//   PLC/PLC Instance <-> EtherCAT Master BKCUCX/TcTerminals210_EK1100_1/TcTerminals210_1BK1250/A_0187(KL 2012, 2 Ch. Output (24V, 0.5 A))
//     PlcTask Outputs/GVL_iXlinker.EtherCAT_Master_BKCUCX.TcTerminals210_EK1100_1.TcTerminals210_1BK1250.A_0187_KL_2012_2_Ch_Output_24V_0_5_A.Channel_1.Output <-> Channel 1/Output
//     PlcTask Outputs/GVL_iXlinker.EtherCAT_Master_BKCUCX.TcTerminals210_EK1100_1.TcTerminals210_1BK1250.A_0187_KL_2012_2_Ch_Output_24V_0_5_A.Channel_2.Output <-> Channel 2/Output
//   PLC/PLC Instance <-> EtherCAT Master BKCUCX/TcTerminals210_EK1100_1/TcTerminals210_1BK1250/A_0188(KL 2022, 2 Ch. Output (24V, 2.0 A))
//     PlcTask Outputs/GVL_iXlinker.EtherCAT_Master_BKCUCX.TcTerminals210_EK1100_1.TcTerminals210_1BK1250.A_0188_KL_2022_2_Ch_Output_24V_2_0_A.Channel_1.Output <-> Channel 1/Output
//     PlcTask Outputs/GVL_iXlinker.EtherCAT_Master_BKCUCX.TcTerminals210_EK1100_1.TcTerminals210_1BK1250.A_0188_KL_2022_2_Ch_Output_24V_2_0_A.Channel_2.Output <-> Channel 2/Output
//   PLC/PLC Instance <-> EtherCAT Master BKCUCX/TcTerminals210_EK1100_1/TcTerminals210_1BK1250/A_0189(KL 2032, 2 Ch. Output with Protection (24V, 0.5 A))
//     PlcTask Outputs/GVL_iXlinker.EtherCAT_Master_BKCUCX.TcTerminals210_EK1100_1.TcTerminals210_1BK1250.A_0189_KL_2032_2_Ch_Output_with_Protection_24V_0_5_A.Channel_1.Output <-> Channel 1/Output
//     PlcTask Outputs/GVL_iXlinker.EtherCAT_Master_BKCUCX.TcTerminals210_EK1100_1.TcTerminals210_1BK1250.A_0189_KL_2032_2_Ch_Output_with_Protection_24V_0_5_A.Channel_2.Output <-> Channel 2/Output
//   PLC/PLC Instance <-> EtherCAT Master BKCUCX/TcTerminals210_EK1100_1/TcTerminals210_1BK1250/A_0190(KL 2114, 4 Ch. Output (24V, 0.5 A))
//     PlcTask Outputs/GVL_iXlinker.EtherCAT_Master_BKCUCX.TcTerminals210_EK1100_1.TcTerminals210_1BK1250.A_0190_KL_2114_4_Ch_Output_24V_0_5_A.Channel_1.Output <-> Channel 1/Output
//     PlcTask Outputs/GVL_iXlinker.EtherCAT_Master_BKCUCX.TcTerminals210_EK1100_1.TcTerminals210_1BK1250.A_0190_KL_2114_4_Ch_Output_24V_0_5_A.Channel_2.Output <-> Channel 2/Output
//     PlcTask Outputs/GVL_iXlinker.EtherCAT_Master_BKCUCX.TcTerminals210_EK1100_1.TcTerminals210_1BK1250.A_0190_KL_2114_4_Ch_Output_24V_0_5_A.Channel_3.Output <-> Channel 3/Output
//     PlcTask Outputs/GVL_iXlinker.EtherCAT_Master_BKCUCX.TcTerminals210_EK1100_1.TcTerminals210_1BK1250.A_0190_KL_2114_4_Ch_Output_24V_0_5_A.Channel_4.Output <-> Channel 4/Output
//   PLC/PLC Instance <-> EtherCAT Master BKCUCX/TcTerminals210_EK1100_1/TcTerminals210_1BK1250/A_0191(KL 2124, 4 Ch. Output (5V, 20 mA))
//     PlcTask Outputs/GVL_iXlinker.EtherCAT_Master_BKCUCX.TcTerminals210_EK1100_1.TcTerminals210_1BK1250.A_0191_KL_2124_4_Ch_Output_5V_20_mA.Channel_1.Output <-> Channel 1/Output
//     PlcTask Outputs/GVL_iXlinker.EtherCAT_Master_BKCUCX.TcTerminals210_EK1100_1.TcTerminals210_1BK1250.A_0191_KL_2124_4_Ch_Output_5V_20_mA.Channel_2.Output <-> Channel 2/Output
//     PlcTask Outputs/GVL_iXlinker.EtherCAT_Master_BKCUCX.TcTerminals210_EK1100_1.TcTerminals210_1BK1250.A_0191_KL_2124_4_Ch_Output_5V_20_mA.Channel_3.Output <-> Channel 3/Output
//     PlcTask Outputs/GVL_iXlinker.EtherCAT_Master_BKCUCX.TcTerminals210_EK1100_1.TcTerminals210_1BK1250.A_0191_KL_2124_4_Ch_Output_5V_20_mA.Channel_4.Output <-> Channel 4/Output
//   PLC/PLC Instance <-> EtherCAT Master BKCUCX/TcTerminals210_EK1100_1/TcTerminals210_1BK1250/A_0192(KL 2134, 4 Ch. Output with Protection (24V, 0.5 A))
//     PlcTask Outputs/GVL_iXlinker.EtherCAT_Master_BKCUCX.TcTerminals210_EK1100_1.TcTerminals210_1BK1250.A_0192_KL_2134_4_Ch_Output_with_Protection_24V_0_5_A.Channel_1.Output <-> Channel 1/Output
//     PlcTask Outputs/GVL_iXlinker.EtherCAT_Master_BKCUCX.TcTerminals210_EK1100_1.TcTerminals210_1BK1250.A_0192_KL_2134_4_Ch_Output_with_Protection_24V_0_5_A.Channel_2.Output <-> Channel 2/Output
//     PlcTask Outputs/GVL_iXlinker.EtherCAT_Master_BKCUCX.TcTerminals210_EK1100_1.TcTerminals210_1BK1250.A_0192_KL_2134_4_Ch_Output_with_Protection_24V_0_5_A.Channel_3.Output <-> Channel 3/Output
//     PlcTask Outputs/GVL_iXlinker.EtherCAT_Master_BKCUCX.TcTerminals210_EK1100_1.TcTerminals210_1BK1250.A_0192_KL_2134_4_Ch_Output_with_Protection_24V_0_5_A.Channel_4.Output <-> Channel 4/Output
//   PLC/PLC Instance <-> EtherCAT Master BKCUCX/TcTerminals210_EK1100_1/TcTerminals210_1BK1250/A_0193(KL 2184, 4 Ch. Output neg. (24V, 0.5 A))
//     PlcTask Outputs/GVL_iXlinker.EtherCAT_Master_BKCUCX.TcTerminals210_EK1100_1.TcTerminals210_1BK1250.A_0193_KL_2184_4_Ch_Output_neg_24V_0_5_A.Channel_1.Output <-> Channel 1/Output
//     PlcTask Outputs/GVL_iXlinker.EtherCAT_Master_BKCUCX.TcTerminals210_EK1100_1.TcTerminals210_1BK1250.A_0193_KL_2184_4_Ch_Output_neg_24V_0_5_A.Channel_2.Output <-> Channel 2/Output
//     PlcTask Outputs/GVL_iXlinker.EtherCAT_Master_BKCUCX.TcTerminals210_EK1100_1.TcTerminals210_1BK1250.A_0193_KL_2184_4_Ch_Output_neg_24V_0_5_A.Channel_3.Output <-> Channel 3/Output
//     PlcTask Outputs/GVL_iXlinker.EtherCAT_Master_BKCUCX.TcTerminals210_EK1100_1.TcTerminals210_1BK1250.A_0193_KL_2184_4_Ch_Output_neg_24V_0_5_A.Channel_4.Output <-> Channel 4/Output
//   PLC/PLC Instance <-> EtherCAT Master BKCUCX/TcTerminals210_EK1100_1/TcTerminals210_1BK1250/A_0194(KL 2212, 2 Ch. Output (24V, 0.5 A with Diag))
//     PlcTask Inputs/GVL_iXlinker.EtherCAT_Master_BKCUCX.TcTerminals210_EK1100_1.TcTerminals210_1BK1250.A_0194_KL_2212_2_Ch_Output_24V_0_5_A_with_Diag.Channel_1.WireBreak <-> Channel 1/WireBreak
//     PlcTask Inputs/GVL_iXlinker.EtherCAT_Master_BKCUCX.TcTerminals210_EK1100_1.TcTerminals210_1BK1250.A_0194_KL_2212_2_Ch_Output_24V_0_5_A_with_Diag.Channel_2.WireBreak <-> Channel 2/WireBreak
//     PlcTask Inputs/GVL_iXlinker.EtherCAT_Master_BKCUCX.TcTerminals210_EK1100_1.TcTerminals210_1BK1250.A_0194_KL_2212_2_Ch_Output_24V_0_5_A_with_Diag.Channel_1.Curcuit <-> Channel 1/Curcuit
//     PlcTask Inputs/GVL_iXlinker.EtherCAT_Master_BKCUCX.TcTerminals210_EK1100_1.TcTerminals210_1BK1250.A_0194_KL_2212_2_Ch_Output_24V_0_5_A_with_Diag.Channel_2.Curcuit <-> Channel 2/Curcuit
//     PlcTask Outputs/GVL_iXlinker.EtherCAT_Master_BKCUCX.TcTerminals210_EK1100_1.TcTerminals210_1BK1250.A_0194_KL_2212_2_Ch_Output_24V_0_5_A_with_Diag.Channel_1.Output <-> Channel 1/Output
//     PlcTask Outputs/GVL_iXlinker.EtherCAT_Master_BKCUCX.TcTerminals210_EK1100_1.TcTerminals210_1BK1250.A_0194_KL_2212_2_Ch_Output_24V_0_5_A_with_Diag.Channel_2.Output <-> Channel 2/Output
//   PLC/PLC Instance <-> EtherCAT Master BKCUCX/TcTerminals210_EK1100_1/TcTerminals210_1BK1250/A_0195(KL 1202, 2 Ch. Input (24V, with Power))
//     PlcTask Inputs/GVL_iXlinker.EtherCAT_Master_BKCUCX.TcTerminals210_EK1100_1.TcTerminals210_1BK1250.A_0195_KL_1202_2_Ch_Input_24V_with_Power.Channel_1.Input <-> Channel 1/Input
//     PlcTask Inputs/GVL_iXlinker.EtherCAT_Master_BKCUCX.TcTerminals210_EK1100_1.TcTerminals210_1BK1250.A_0195_KL_1202_2_Ch_Input_24V_with_Power.Channel_2.Input <-> Channel 2/Input
//     PlcTask Inputs/GVL_iXlinker.EtherCAT_Master_BKCUCX.TcTerminals210_EK1100_1.TcTerminals210_1BK1250.A_0195_KL_1202_2_Ch_Input_24V_with_Power.Channel_1.Error <-> Channel 1/Error
//     PlcTask Inputs/GVL_iXlinker.EtherCAT_Master_BKCUCX.TcTerminals210_EK1100_1.TcTerminals210_1BK1250.A_0195_KL_1202_2_Ch_Input_24V_with_Power.Channel_2.Error <-> Channel 2/Error
//     PlcTask Outputs/GVL_iXlinker.EtherCAT_Master_BKCUCX.TcTerminals210_EK1100_1.TcTerminals210_1BK1250.A_0195_KL_1202_2_Ch_Input_24V_with_Power.Channel_1.Power <-> Channel 1/Power
//     PlcTask Outputs/GVL_iXlinker.EtherCAT_Master_BKCUCX.TcTerminals210_EK1100_1.TcTerminals210_1BK1250.A_0195_KL_1202_2_Ch_Input_24V_with_Power.Channel_2.Power <-> Channel 2/Power
//   PLC/PLC Instance <-> EtherCAT Master BKCUCX/TcTerminals210_EK1100_1/TcTerminals210_1BK1250/A_0196(KL 2404, 4 Ch. Output with Protection (24V, 0.5 A, 2 wire))
//     PlcTask Outputs/GVL_iXlinker.EtherCAT_Master_BKCUCX.TcTerminals210_EK1100_1.TcTerminals210_1BK1250.A_0196_KL_2404_4_Ch_Output_with_Protection_24V_0_5_A_2_wire.Channel_1.Output <-> Channel 1/Output
//     PlcTask Outputs/GVL_iXlinker.EtherCAT_Master_BKCUCX.TcTerminals210_EK1100_1.TcTerminals210_1BK1250.A_0196_KL_2404_4_Ch_Output_with_Protection_24V_0_5_A_2_wire.Channel_2.Output <-> Channel 2/Output
//     PlcTask Outputs/GVL_iXlinker.EtherCAT_Master_BKCUCX.TcTerminals210_EK1100_1.TcTerminals210_1BK1250.A_0196_KL_2404_4_Ch_Output_with_Protection_24V_0_5_A_2_wire.Channel_3.Output <-> Channel 3/Output
//     PlcTask Outputs/GVL_iXlinker.EtherCAT_Master_BKCUCX.TcTerminals210_EK1100_1.TcTerminals210_1BK1250.A_0196_KL_2404_4_Ch_Output_with_Protection_24V_0_5_A_2_wire.Channel_4.Output <-> Channel 4/Output
//   PLC/PLC Instance <-> EtherCAT Master BKCUCX/TcTerminals210_EK1100_1/TcTerminals210_1BK1250/A_0197(KL 2408, 8 Ch. Output (24V, 0.5 A, 3 A max))
//     PlcTask Outputs/GVL_iXlinker.EtherCAT_Master_BKCUCX.TcTerminals210_EK1100_1.TcTerminals210_1BK1250.A_0197_KL_2408_8_Ch_Output_24V_0_5_A_3_A_max.Channel_1.Output <-> Channel 1/Output
//     PlcTask Outputs/GVL_iXlinker.EtherCAT_Master_BKCUCX.TcTerminals210_EK1100_1.TcTerminals210_1BK1250.A_0197_KL_2408_8_Ch_Output_24V_0_5_A_3_A_max.Channel_2.Output <-> Channel 2/Output
//     PlcTask Outputs/GVL_iXlinker.EtherCAT_Master_BKCUCX.TcTerminals210_EK1100_1.TcTerminals210_1BK1250.A_0197_KL_2408_8_Ch_Output_24V_0_5_A_3_A_max.Channel_3.Output <-> Channel 3/Output
//     PlcTask Outputs/GVL_iXlinker.EtherCAT_Master_BKCUCX.TcTerminals210_EK1100_1.TcTerminals210_1BK1250.A_0197_KL_2408_8_Ch_Output_24V_0_5_A_3_A_max.Channel_4.Output <-> Channel 4/Output
//     PlcTask Outputs/GVL_iXlinker.EtherCAT_Master_BKCUCX.TcTerminals210_EK1100_1.TcTerminals210_1BK1250.A_0197_KL_2408_8_Ch_Output_24V_0_5_A_3_A_max.Channel_5.Output <-> Channel 5/Output
//     PlcTask Outputs/GVL_iXlinker.EtherCAT_Master_BKCUCX.TcTerminals210_EK1100_1.TcTerminals210_1BK1250.A_0197_KL_2408_8_Ch_Output_24V_0_5_A_3_A_max.Channel_6.Output <-> Channel 6/Output
//     PlcTask Outputs/GVL_iXlinker.EtherCAT_Master_BKCUCX.TcTerminals210_EK1100_1.TcTerminals210_1BK1250.A_0197_KL_2408_8_Ch_Output_24V_0_5_A_3_A_max.Channel_7.Output <-> Channel 7/Output
//     PlcTask Outputs/GVL_iXlinker.EtherCAT_Master_BKCUCX.TcTerminals210_EK1100_1.TcTerminals210_1BK1250.A_0197_KL_2408_8_Ch_Output_24V_0_5_A_3_A_max.Channel_8.Output <-> Channel 8/Output
//   PLC/PLC Instance <-> EtherCAT Master BKCUCX/TcTerminals210_EK1100_1/TcTerminals210_1BK1250/A_0198(KL 2424, 4 Ch. Output with Protection (24V, 2 A, 2 wire))
//     PlcTask Outputs/GVL_iXlinker.EtherCAT_Master_BKCUCX.TcTerminals210_EK1100_1.TcTerminals210_1BK1250.A_0198_KL_2424_4_Ch_Output_with_Protection_24V_2_A_2_wire.Channel_1.Output <-> Channel 1/Output
//     PlcTask Outputs/GVL_iXlinker.EtherCAT_Master_BKCUCX.TcTerminals210_EK1100_1.TcTerminals210_1BK1250.A_0198_KL_2424_4_Ch_Output_with_Protection_24V_2_A_2_wire.Channel_2.Output <-> Channel 2/Output
//     PlcTask Outputs/GVL_iXlinker.EtherCAT_Master_BKCUCX.TcTerminals210_EK1100_1.TcTerminals210_1BK1250.A_0198_KL_2424_4_Ch_Output_with_Protection_24V_2_A_2_wire.Channel_3.Output <-> Channel 3/Output
//     PlcTask Outputs/GVL_iXlinker.EtherCAT_Master_BKCUCX.TcTerminals210_EK1100_1.TcTerminals210_1BK1250.A_0198_KL_2424_4_Ch_Output_with_Protection_24V_2_A_2_wire.Channel_4.Output <-> Channel 4/Output
//   PLC/PLC Instance <-> EtherCAT Master BKCUCX/TcTerminals210_EK1100_1/TcTerminals210_1BK1250/A_0199(KL 2442, 2 Ch. Output (24V, 8 A, 8 A max))
//     PlcTask Outputs/GVL_iXlinker.EtherCAT_Master_BKCUCX.TcTerminals210_EK1100_1.TcTerminals210_1BK1250.A_0199_KL_2442_2_Ch_Output_24V_8_A_8_A_max.Channel_1.Output <-> Channel 1/Output
//     PlcTask Outputs/GVL_iXlinker.EtherCAT_Master_BKCUCX.TcTerminals210_EK1100_1.TcTerminals210_1BK1250.A_0199_KL_2442_2_Ch_Output_24V_8_A_8_A_max.Channel_2.Output <-> Channel 2/Output
//   PLC/PLC Instance <-> EtherCAT Master BKCUCX/TcTerminals210_EK1100_1/TcTerminals210_1BK1250/A_0200(KL 2488, 8 Ch. Output (24V neg, 0.5 A, 3 A max))
//     PlcTask Outputs/GVL_iXlinker.EtherCAT_Master_BKCUCX.TcTerminals210_EK1100_1.TcTerminals210_1BK1250.A_0200_KL_2488_8_Ch_Output_24V_neg_0_5_A_3_A_max.Channel_1.Output <-> Channel 1/Output
//     PlcTask Outputs/GVL_iXlinker.EtherCAT_Master_BKCUCX.TcTerminals210_EK1100_1.TcTerminals210_1BK1250.A_0200_KL_2488_8_Ch_Output_24V_neg_0_5_A_3_A_max.Channel_2.Output <-> Channel 2/Output
//     PlcTask Outputs/GVL_iXlinker.EtherCAT_Master_BKCUCX.TcTerminals210_EK1100_1.TcTerminals210_1BK1250.A_0200_KL_2488_8_Ch_Output_24V_neg_0_5_A_3_A_max.Channel_3.Output <-> Channel 3/Output
//     PlcTask Outputs/GVL_iXlinker.EtherCAT_Master_BKCUCX.TcTerminals210_EK1100_1.TcTerminals210_1BK1250.A_0200_KL_2488_8_Ch_Output_24V_neg_0_5_A_3_A_max.Channel_4.Output <-> Channel 4/Output
//     PlcTask Outputs/GVL_iXlinker.EtherCAT_Master_BKCUCX.TcTerminals210_EK1100_1.TcTerminals210_1BK1250.A_0200_KL_2488_8_Ch_Output_24V_neg_0_5_A_3_A_max.Channel_5.Output <-> Channel 5/Output
//     PlcTask Outputs/GVL_iXlinker.EtherCAT_Master_BKCUCX.TcTerminals210_EK1100_1.TcTerminals210_1BK1250.A_0200_KL_2488_8_Ch_Output_24V_neg_0_5_A_3_A_max.Channel_6.Output <-> Channel 6/Output
//     PlcTask Outputs/GVL_iXlinker.EtherCAT_Master_BKCUCX.TcTerminals210_EK1100_1.TcTerminals210_1BK1250.A_0200_KL_2488_8_Ch_Output_24V_neg_0_5_A_3_A_max.Channel_7.Output <-> Channel 7/Output
//     PlcTask Outputs/GVL_iXlinker.EtherCAT_Master_BKCUCX.TcTerminals210_EK1100_1.TcTerminals210_1BK1250.A_0200_KL_2488_8_Ch_Output_24V_neg_0_5_A_3_A_max.Channel_8.Output <-> Channel 8/Output
//   PLC/PLC Instance <-> EtherCAT Master BKCUCX/TcTerminals210_EK1100_1/TcTerminals210_1BK1250/A_0201(KL 2284, 4 Ch. Output (24V, 2 A, reverse switching))
//     PlcTask Outputs/GVL_iXlinker.EtherCAT_Master_BKCUCX.TcTerminals210_EK1100_1.TcTerminals210_1BK1250.A_0201_KL_2284_4_Ch_Output_24V_2_A_reverse_switching.Channel_1.CW <-> Channel 1/CW
//     PlcTask Outputs/GVL_iXlinker.EtherCAT_Master_BKCUCX.TcTerminals210_EK1100_1.TcTerminals210_1BK1250.A_0201_KL_2284_4_Ch_Output_24V_2_A_reverse_switching.Channel_2.CW <-> Channel 2/CW
//     PlcTask Outputs/GVL_iXlinker.EtherCAT_Master_BKCUCX.TcTerminals210_EK1100_1.TcTerminals210_1BK1250.A_0201_KL_2284_4_Ch_Output_24V_2_A_reverse_switching.Channel_3.CW <-> Channel 3/CW
//     PlcTask Outputs/GVL_iXlinker.EtherCAT_Master_BKCUCX.TcTerminals210_EK1100_1.TcTerminals210_1BK1250.A_0201_KL_2284_4_Ch_Output_24V_2_A_reverse_switching.Channel_4.CW <-> Channel 4/CW
//     PlcTask Outputs/GVL_iXlinker.EtherCAT_Master_BKCUCX.TcTerminals210_EK1100_1.TcTerminals210_1BK1250.A_0201_KL_2284_4_Ch_Output_24V_2_A_reverse_switching.Channel_1.CCW <-> Channel 1/CCW
//     PlcTask Outputs/GVL_iXlinker.EtherCAT_Master_BKCUCX.TcTerminals210_EK1100_1.TcTerminals210_1BK1250.A_0201_KL_2284_4_Ch_Output_24V_2_A_reverse_switching.Channel_2.CCW <-> Channel 2/CCW
//     PlcTask Outputs/GVL_iXlinker.EtherCAT_Master_BKCUCX.TcTerminals210_EK1100_1.TcTerminals210_1BK1250.A_0201_KL_2284_4_Ch_Output_24V_2_A_reverse_switching.Channel_3.CCW <-> Channel 3/CCW
//     PlcTask Outputs/GVL_iXlinker.EtherCAT_Master_BKCUCX.TcTerminals210_EK1100_1.TcTerminals210_1BK1250.A_0201_KL_2284_4_Ch_Output_24V_2_A_reverse_switching.Channel_4.CCW <-> Channel 4/CCW
//   PLC/PLC Instance <-> EtherCAT Master BKCUCX/TcTerminals210_EK1100_1/TcTerminals210_1BK1250/A_0202(KL 2502, 2 Ch. PWM Output 24V)
//     PlcTask Inputs/GVL_iXlinker.EtherCAT_Master_BKCUCX.TcTerminals210_EK1100_1.TcTerminals210_1BK1250.A_0202_KL_2502_2_Ch_PWM_Output_24V.Channel_1.State <-> Channel 1/State
//     PlcTask Inputs/GVL_iXlinker.EtherCAT_Master_BKCUCX.TcTerminals210_EK1100_1.TcTerminals210_1BK1250.A_0202_KL_2502_2_Ch_PWM_Output_24V.Channel_2.State <-> Channel 2/State
//     PlcTask Inputs/GVL_iXlinker.EtherCAT_Master_BKCUCX.TcTerminals210_EK1100_1.TcTerminals210_1BK1250.A_0202_KL_2502_2_Ch_PWM_Output_24V.Channel_1.Data_In <-> Channel 1/Data In
//     PlcTask Inputs/GVL_iXlinker.EtherCAT_Master_BKCUCX.TcTerminals210_EK1100_1.TcTerminals210_1BK1250.A_0202_KL_2502_2_Ch_PWM_Output_24V.Channel_2.Data_In <-> Channel 2/Data In
//     PlcTask Outputs/GVL_iXlinker.EtherCAT_Master_BKCUCX.TcTerminals210_EK1100_1.TcTerminals210_1BK1250.A_0202_KL_2502_2_Ch_PWM_Output_24V.Channel_1.Ctrl <-> Channel 1/Ctrl
//     PlcTask Outputs/GVL_iXlinker.EtherCAT_Master_BKCUCX.TcTerminals210_EK1100_1.TcTerminals210_1BK1250.A_0202_KL_2502_2_Ch_PWM_Output_24V.Channel_2.Ctrl <-> Channel 2/Ctrl
//     PlcTask Outputs/GVL_iXlinker.EtherCAT_Master_BKCUCX.TcTerminals210_EK1100_1.TcTerminals210_1BK1250.A_0202_KL_2502_2_Ch_PWM_Output_24V.Channel_1.Data_Out <-> Channel 1/Data Out
//     PlcTask Outputs/GVL_iXlinker.EtherCAT_Master_BKCUCX.TcTerminals210_EK1100_1.TcTerminals210_1BK1250.A_0202_KL_2502_2_Ch_PWM_Output_24V.Channel_2.Data_Out <-> Channel 2/Data Out
//   PLC/PLC Instance <-> EtherCAT Master BKCUCX/TcTerminals210_EK1100_1/TcTerminals210_1BK1250/A_0203(KL 2512, 2 Ch. PWM Output (24V, 1,5A, neg))
//     PlcTask Inputs/GVL_iXlinker.EtherCAT_Master_BKCUCX.TcTerminals210_EK1100_1.TcTerminals210_1BK1250.A_0203_KL_2512_2_Ch_PWM_Output_24V_1_5A_neg.Channel_1.State <-> Channel 1/State
//     PlcTask Inputs/GVL_iXlinker.EtherCAT_Master_BKCUCX.TcTerminals210_EK1100_1.TcTerminals210_1BK1250.A_0203_KL_2512_2_Ch_PWM_Output_24V_1_5A_neg.Channel_2.State <-> Channel 2/State
//     PlcTask Inputs/GVL_iXlinker.EtherCAT_Master_BKCUCX.TcTerminals210_EK1100_1.TcTerminals210_1BK1250.A_0203_KL_2512_2_Ch_PWM_Output_24V_1_5A_neg.Channel_1.Data_In <-> Channel 1/Data In
//     PlcTask Inputs/GVL_iXlinker.EtherCAT_Master_BKCUCX.TcTerminals210_EK1100_1.TcTerminals210_1BK1250.A_0203_KL_2512_2_Ch_PWM_Output_24V_1_5A_neg.Channel_2.Data_In <-> Channel 2/Data In
//     PlcTask Outputs/GVL_iXlinker.EtherCAT_Master_BKCUCX.TcTerminals210_EK1100_1.TcTerminals210_1BK1250.A_0203_KL_2512_2_Ch_PWM_Output_24V_1_5A_neg.Channel_1.Ctrl <-> Channel 1/Ctrl
//     PlcTask Outputs/GVL_iXlinker.EtherCAT_Master_BKCUCX.TcTerminals210_EK1100_1.TcTerminals210_1BK1250.A_0203_KL_2512_2_Ch_PWM_Output_24V_1_5A_neg.Channel_2.Ctrl <-> Channel 2/Ctrl
//     PlcTask Outputs/GVL_iXlinker.EtherCAT_Master_BKCUCX.TcTerminals210_EK1100_1.TcTerminals210_1BK1250.A_0203_KL_2512_2_Ch_PWM_Output_24V_1_5A_neg.Channel_1.Data_Out <-> Channel 1/Data Out
//     PlcTask Outputs/GVL_iXlinker.EtherCAT_Master_BKCUCX.TcTerminals210_EK1100_1.TcTerminals210_1BK1250.A_0203_KL_2512_2_Ch_PWM_Output_24V_1_5A_neg.Channel_2.Data_Out <-> Channel 2/Data Out
//   PLC/PLC Instance <-> EtherCAT Master BKCUCX/TcTerminals210_EK1100_1/TcTerminals210_1BK1250/A_0204(KL 2521, 1 Ch. Pulse Train Output)
//     PlcTask Inputs/GVL_iXlinker.EtherCAT_Master_BKCUCX.TcTerminals210_EK1100_1.TcTerminals210_1BK1250.A_0204_KL_2521_1_Ch_Pulse_Train_Output.Channel_1.State <-> Channel 1/State
//     PlcTask Inputs/GVL_iXlinker.EtherCAT_Master_BKCUCX.TcTerminals210_EK1100_1.TcTerminals210_1BK1250.A_0204_KL_2521_1_Ch_Pulse_Train_Output.Channel_1.Data_In <-> Channel 1/Data In
//     PlcTask Outputs/GVL_iXlinker.EtherCAT_Master_BKCUCX.TcTerminals210_EK1100_1.TcTerminals210_1BK1250.A_0204_KL_2521_1_Ch_Pulse_Train_Output.Channel_1.Ctrl <-> Channel 1/Ctrl
//     PlcTask Outputs/GVL_iXlinker.EtherCAT_Master_BKCUCX.TcTerminals210_EK1100_1.TcTerminals210_1BK1250.A_0204_KL_2521_1_Ch_Pulse_Train_Output.Channel_1.Data_Out <-> Channel 1/Data Out
//   PLC/PLC Instance <-> EtherCAT Master BKCUCX/TcTerminals210_EK1100_1/TcTerminals210_1BK1250/A_0205(KL 2531, 1 Ch. Stepper (24V, 1.5 A))
//     PlcTask Inputs/GVL_iXlinker.EtherCAT_Master_BKCUCX.TcTerminals210_EK1100_1.TcTerminals210_1BK1250.A_0205_KL_2531_1_Ch_Stepper_24V_1_5_A.Channel_1.Status <-> Channel 1/Status
//     PlcTask Inputs/GVL_iXlinker.EtherCAT_Master_BKCUCX.TcTerminals210_EK1100_1.TcTerminals210_1BK1250.A_0205_KL_2531_1_Ch_Stepper_24V_1_5_A.Channel_1.Position <-> Channel 1/Position
//     PlcTask Inputs/GVL_iXlinker.EtherCAT_Master_BKCUCX.TcTerminals210_EK1100_1.TcTerminals210_1BK1250.A_0205_KL_2531_1_Ch_Stepper_24V_1_5_A.Channel_1.ExtStatus <-> Channel 1/ExtStatus
//     PlcTask Outputs/GVL_iXlinker.EtherCAT_Master_BKCUCX.TcTerminals210_EK1100_1.TcTerminals210_1BK1250.A_0205_KL_2531_1_Ch_Stepper_24V_1_5_A.Channel_1.Ctrl <-> Channel 1/Ctrl
//     PlcTask Outputs/GVL_iXlinker.EtherCAT_Master_BKCUCX.TcTerminals210_EK1100_1.TcTerminals210_1BK1250.A_0205_KL_2531_1_Ch_Stepper_24V_1_5_A.Channel_1.Velocity <-> Channel 1/Velocity
//     PlcTask Outputs/GVL_iXlinker.EtherCAT_Master_BKCUCX.TcTerminals210_EK1100_1.TcTerminals210_1BK1250.A_0205_KL_2531_1_Ch_Stepper_24V_1_5_A.Channel_1.ExtCtrl <-> Channel 1/ExtCtrl
//   PLC/PLC Instance <-> EtherCAT Master BKCUCX/TcTerminals210_EK1100_1/TcTerminals210_1BK1250/A_0206(KL 2531-1000, 1 Ch. Stepper (24V, 1.5 A))
//     PlcTask Inputs/GVL_iXlinker.EtherCAT_Master_BKCUCX.TcTerminals210_EK1100_1.TcTerminals210_1BK1250.A_0206_KL_2531_1000_1_Ch_Stepper_24V_1_5_A.Channel_1.Status <-> Channel 1/Status
//     PlcTask Inputs/GVL_iXlinker.EtherCAT_Master_BKCUCX.TcTerminals210_EK1100_1.TcTerminals210_1BK1250.A_0206_KL_2531_1000_1_Ch_Stepper_24V_1_5_A.Channel_1.Position <-> Channel 1/Position
//     PlcTask Inputs/GVL_iXlinker.EtherCAT_Master_BKCUCX.TcTerminals210_EK1100_1.TcTerminals210_1BK1250.A_0206_KL_2531_1000_1_Ch_Stepper_24V_1_5_A.Channel_1.ExtStatus <-> Channel 1/ExtStatus
//     PlcTask Outputs/GVL_iXlinker.EtherCAT_Master_BKCUCX.TcTerminals210_EK1100_1.TcTerminals210_1BK1250.A_0206_KL_2531_1000_1_Ch_Stepper_24V_1_5_A.Channel_1.Ctrl <-> Channel 1/Ctrl
//     PlcTask Outputs/GVL_iXlinker.EtherCAT_Master_BKCUCX.TcTerminals210_EK1100_1.TcTerminals210_1BK1250.A_0206_KL_2531_1000_1_Ch_Stepper_24V_1_5_A.Channel_1.Velocity <-> Channel 1/Velocity
//     PlcTask Outputs/GVL_iXlinker.EtherCAT_Master_BKCUCX.TcTerminals210_EK1100_1.TcTerminals210_1BK1250.A_0206_KL_2531_1000_1_Ch_Stepper_24V_1_5_A.Channel_1.ExtCtrl <-> Channel 1/ExtCtrl
//   PLC/PLC Instance <-> EtherCAT Master BKCUCX/TcTerminals210_EK1100_1/TcTerminals210_1BK1250/A_0207(KL 2532, 2 Ch. DC Amplifier (24V, 1 A))
//     PlcTask Inputs/GVL_iXlinker.EtherCAT_Master_BKCUCX.TcTerminals210_EK1100_1.TcTerminals210_1BK1250.A_0207_KL_2532_2_Ch_DC_Amplifier_24V_1_A.Channel_1.State <-> Channel 1/State
//     PlcTask Inputs/GVL_iXlinker.EtherCAT_Master_BKCUCX.TcTerminals210_EK1100_1.TcTerminals210_1BK1250.A_0207_KL_2532_2_Ch_DC_Amplifier_24V_1_A.Channel_2.State <-> Channel 2/State
//     PlcTask Inputs/GVL_iXlinker.EtherCAT_Master_BKCUCX.TcTerminals210_EK1100_1.TcTerminals210_1BK1250.A_0207_KL_2532_2_Ch_DC_Amplifier_24V_1_A.Channel_1.Data_In <-> Channel 1/Data In
//     PlcTask Inputs/GVL_iXlinker.EtherCAT_Master_BKCUCX.TcTerminals210_EK1100_1.TcTerminals210_1BK1250.A_0207_KL_2532_2_Ch_DC_Amplifier_24V_1_A.Channel_2.Data_In <-> Channel 2/Data In
//     PlcTask Outputs/GVL_iXlinker.EtherCAT_Master_BKCUCX.TcTerminals210_EK1100_1.TcTerminals210_1BK1250.A_0207_KL_2532_2_Ch_DC_Amplifier_24V_1_A.Channel_1.Ctrl <-> Channel 1/Ctrl
//     PlcTask Outputs/GVL_iXlinker.EtherCAT_Master_BKCUCX.TcTerminals210_EK1100_1.TcTerminals210_1BK1250.A_0207_KL_2532_2_Ch_DC_Amplifier_24V_1_A.Channel_2.Ctrl <-> Channel 2/Ctrl
//     PlcTask Outputs/GVL_iXlinker.EtherCAT_Master_BKCUCX.TcTerminals210_EK1100_1.TcTerminals210_1BK1250.A_0207_KL_2532_2_Ch_DC_Amplifier_24V_1_A.Channel_1.Data_Out <-> Channel 1/Data Out
//     PlcTask Outputs/GVL_iXlinker.EtherCAT_Master_BKCUCX.TcTerminals210_EK1100_1.TcTerminals210_1BK1250.A_0207_KL_2532_2_Ch_DC_Amplifier_24V_1_A.Channel_2.Data_Out <-> Channel 2/Data Out
//   PLC/PLC Instance <-> EtherCAT Master BKCUCX/TcTerminals210_EK1100_1/TcTerminals210_1BK1250/A_0208(KL 2535, 2 Ch. PWM Amplifier (24V, 1 A))
//     PlcTask Inputs/GVL_iXlinker.EtherCAT_Master_BKCUCX.TcTerminals210_EK1100_1.TcTerminals210_1BK1250.A_0208_KL_2535_2_Ch_PWM_Amplifier_24V_1_A.Channel_1.State <-> Channel 1/State
//     PlcTask Inputs/GVL_iXlinker.EtherCAT_Master_BKCUCX.TcTerminals210_EK1100_1.TcTerminals210_1BK1250.A_0208_KL_2535_2_Ch_PWM_Amplifier_24V_1_A.Channel_2.State <-> Channel 2/State
//     PlcTask Inputs/GVL_iXlinker.EtherCAT_Master_BKCUCX.TcTerminals210_EK1100_1.TcTerminals210_1BK1250.A_0208_KL_2535_2_Ch_PWM_Amplifier_24V_1_A.Channel_1.Data_In <-> Channel 1/Data In
//     PlcTask Inputs/GVL_iXlinker.EtherCAT_Master_BKCUCX.TcTerminals210_EK1100_1.TcTerminals210_1BK1250.A_0208_KL_2535_2_Ch_PWM_Amplifier_24V_1_A.Channel_2.Data_In <-> Channel 2/Data In
//     PlcTask Outputs/GVL_iXlinker.EtherCAT_Master_BKCUCX.TcTerminals210_EK1100_1.TcTerminals210_1BK1250.A_0208_KL_2535_2_Ch_PWM_Amplifier_24V_1_A.Channel_1.Ctrl <-> Channel 1/Ctrl
//     PlcTask Outputs/GVL_iXlinker.EtherCAT_Master_BKCUCX.TcTerminals210_EK1100_1.TcTerminals210_1BK1250.A_0208_KL_2535_2_Ch_PWM_Amplifier_24V_1_A.Channel_2.Ctrl <-> Channel 2/Ctrl
//     PlcTask Outputs/GVL_iXlinker.EtherCAT_Master_BKCUCX.TcTerminals210_EK1100_1.TcTerminals210_1BK1250.A_0208_KL_2535_2_Ch_PWM_Amplifier_24V_1_A.Channel_1.Data_Out <-> Channel 1/Data Out
//     PlcTask Outputs/GVL_iXlinker.EtherCAT_Master_BKCUCX.TcTerminals210_EK1100_1.TcTerminals210_1BK1250.A_0208_KL_2535_2_Ch_PWM_Amplifier_24V_1_A.Channel_2.Data_Out <-> Channel 2/Data Out
//   PLC/PLC Instance <-> EtherCAT Master BKCUCX/TcTerminals210_EK1100_1/TcTerminals210_1BK1250/A_0210(KL 2541, 1 Ch. Stepper (50V, 5 A))
//     PlcTask Inputs/GVL_iXlinker.EtherCAT_Master_BKCUCX.TcTerminals210_EK1100_1.TcTerminals210_1BK1250.A_0210_KL_2541_1_Ch_Stepper_50V_5_A.Channel_1.Status <-> Channel 1/Status
//     PlcTask Inputs/GVL_iXlinker.EtherCAT_Master_BKCUCX.TcTerminals210_EK1100_1.TcTerminals210_1BK1250.A_0210_KL_2541_1_Ch_Stepper_50V_5_A.Channel_1.Position <-> Channel 1/Position
//     PlcTask Inputs/GVL_iXlinker.EtherCAT_Master_BKCUCX.TcTerminals210_EK1100_1.TcTerminals210_1BK1250.A_0210_KL_2541_1_Ch_Stepper_50V_5_A.Channel_1.ExtStatus <-> Channel 1/ExtStatus
//     PlcTask Outputs/GVL_iXlinker.EtherCAT_Master_BKCUCX.TcTerminals210_EK1100_1.TcTerminals210_1BK1250.A_0210_KL_2541_1_Ch_Stepper_50V_5_A.Channel_1.Ctrl <-> Channel 1/Ctrl
//     PlcTask Outputs/GVL_iXlinker.EtherCAT_Master_BKCUCX.TcTerminals210_EK1100_1.TcTerminals210_1BK1250.A_0210_KL_2541_1_Ch_Stepper_50V_5_A.Channel_1.Velocity <-> Channel 1/Velocity
//     PlcTask Outputs/GVL_iXlinker.EtherCAT_Master_BKCUCX.TcTerminals210_EK1100_1.TcTerminals210_1BK1250.A_0210_KL_2541_1_Ch_Stepper_50V_5_A.Channel_1.ExtCtrl <-> Channel 1/ExtCtrl
//   PLC/PLC Instance <-> EtherCAT Master BKCUCX/TcTerminals210_EK1100_1/TcTerminals210_1BK1250/A_0211(KL 2541-1000, 1 Ch. Stepper (50V, 5 A))
//     PlcTask Inputs/GVL_iXlinker.EtherCAT_Master_BKCUCX.TcTerminals210_EK1100_1.TcTerminals210_1BK1250.A_0211_KL_2541_1000_1_Ch_Stepper_50V_5_A.Channel_1.Status <-> Channel 1/Status
//     PlcTask Inputs/GVL_iXlinker.EtherCAT_Master_BKCUCX.TcTerminals210_EK1100_1.TcTerminals210_1BK1250.A_0211_KL_2541_1000_1_Ch_Stepper_50V_5_A.Channel_1.Position <-> Channel 1/Position
//     PlcTask Inputs/GVL_iXlinker.EtherCAT_Master_BKCUCX.TcTerminals210_EK1100_1.TcTerminals210_1BK1250.A_0211_KL_2541_1000_1_Ch_Stepper_50V_5_A.Channel_1.ExtStatus <-> Channel 1/ExtStatus
//     PlcTask Outputs/GVL_iXlinker.EtherCAT_Master_BKCUCX.TcTerminals210_EK1100_1.TcTerminals210_1BK1250.A_0211_KL_2541_1000_1_Ch_Stepper_50V_5_A.Channel_1.Ctrl <-> Channel 1/Ctrl
//     PlcTask Outputs/GVL_iXlinker.EtherCAT_Master_BKCUCX.TcTerminals210_EK1100_1.TcTerminals210_1BK1250.A_0211_KL_2541_1000_1_Ch_Stepper_50V_5_A.Channel_1.Velocity <-> Channel 1/Velocity
//     PlcTask Outputs/GVL_iXlinker.EtherCAT_Master_BKCUCX.TcTerminals210_EK1100_1.TcTerminals210_1BK1250.A_0211_KL_2541_1000_1_Ch_Stepper_50V_5_A.Channel_1.ExtCtrl <-> Channel 1/ExtCtrl
//   PLC/PLC Instance <-> EtherCAT Master BKCUCX/TcTerminals210_EK1100_1/TcTerminals210_1BK1250/A_0212(KL 2542, 2 Ch. DC Amplifier (50V, 3.5 A))
//     PlcTask Inputs/GVL_iXlinker.EtherCAT_Master_BKCUCX.TcTerminals210_EK1100_1.TcTerminals210_1BK1250.A_0212_KL_2542_2_Ch_DC_Amplifier_50V_3_5_A.Channel_1.State <-> Channel 1/State
//     PlcTask Inputs/GVL_iXlinker.EtherCAT_Master_BKCUCX.TcTerminals210_EK1100_1.TcTerminals210_1BK1250.A_0212_KL_2542_2_Ch_DC_Amplifier_50V_3_5_A.Channel_2.State <-> Channel 2/State
//     PlcTask Inputs/GVL_iXlinker.EtherCAT_Master_BKCUCX.TcTerminals210_EK1100_1.TcTerminals210_1BK1250.A_0212_KL_2542_2_Ch_DC_Amplifier_50V_3_5_A.Channel_1.Data_In <-> Channel 1/Data In
//     PlcTask Inputs/GVL_iXlinker.EtherCAT_Master_BKCUCX.TcTerminals210_EK1100_1.TcTerminals210_1BK1250.A_0212_KL_2542_2_Ch_DC_Amplifier_50V_3_5_A.Channel_2.Data_In <-> Channel 2/Data In
//     PlcTask Outputs/GVL_iXlinker.EtherCAT_Master_BKCUCX.TcTerminals210_EK1100_1.TcTerminals210_1BK1250.A_0212_KL_2542_2_Ch_DC_Amplifier_50V_3_5_A.Channel_1.Ctrl <-> Channel 1/Ctrl
//     PlcTask Outputs/GVL_iXlinker.EtherCAT_Master_BKCUCX.TcTerminals210_EK1100_1.TcTerminals210_1BK1250.A_0212_KL_2542_2_Ch_DC_Amplifier_50V_3_5_A.Channel_2.Ctrl <-> Channel 2/Ctrl
//     PlcTask Outputs/GVL_iXlinker.EtherCAT_Master_BKCUCX.TcTerminals210_EK1100_1.TcTerminals210_1BK1250.A_0212_KL_2542_2_Ch_DC_Amplifier_50V_3_5_A.Channel_1.Data_Out <-> Channel 1/Data Out
//     PlcTask Outputs/GVL_iXlinker.EtherCAT_Master_BKCUCX.TcTerminals210_EK1100_1.TcTerminals210_1BK1250.A_0212_KL_2542_2_Ch_DC_Amplifier_50V_3_5_A.Channel_2.Data_Out <-> Channel 2/Data Out
//   PLC/PLC Instance <-> EtherCAT Master BKCUCX/TcTerminals210_EK1100_1/TcTerminals210_1BK1250/A_0213(KL 2545, 2 Ch. PWM Amplifier (50V, 3,5 A))
//     PlcTask Inputs/GVL_iXlinker.EtherCAT_Master_BKCUCX.TcTerminals210_EK1100_1.TcTerminals210_1BK1250.A_0213_KL_2545_2_Ch_PWM_Amplifier_50V_3_5_A.Channel_1.State <-> Channel 1/State
//     PlcTask Inputs/GVL_iXlinker.EtherCAT_Master_BKCUCX.TcTerminals210_EK1100_1.TcTerminals210_1BK1250.A_0213_KL_2545_2_Ch_PWM_Amplifier_50V_3_5_A.Channel_2.State <-> Channel 2/State
//     PlcTask Inputs/GVL_iXlinker.EtherCAT_Master_BKCUCX.TcTerminals210_EK1100_1.TcTerminals210_1BK1250.A_0213_KL_2545_2_Ch_PWM_Amplifier_50V_3_5_A.Channel_1.Data_In <-> Channel 1/Data In
//     PlcTask Inputs/GVL_iXlinker.EtherCAT_Master_BKCUCX.TcTerminals210_EK1100_1.TcTerminals210_1BK1250.A_0213_KL_2545_2_Ch_PWM_Amplifier_50V_3_5_A.Channel_2.Data_In <-> Channel 2/Data In
//     PlcTask Outputs/GVL_iXlinker.EtherCAT_Master_BKCUCX.TcTerminals210_EK1100_1.TcTerminals210_1BK1250.A_0213_KL_2545_2_Ch_PWM_Amplifier_50V_3_5_A.Channel_1.Ctrl <-> Channel 1/Ctrl
//     PlcTask Outputs/GVL_iXlinker.EtherCAT_Master_BKCUCX.TcTerminals210_EK1100_1.TcTerminals210_1BK1250.A_0213_KL_2545_2_Ch_PWM_Amplifier_50V_3_5_A.Channel_2.Ctrl <-> Channel 2/Ctrl
//     PlcTask Outputs/GVL_iXlinker.EtherCAT_Master_BKCUCX.TcTerminals210_EK1100_1.TcTerminals210_1BK1250.A_0213_KL_2545_2_Ch_PWM_Amplifier_50V_3_5_A.Channel_1.Data_Out <-> Channel 1/Data Out
//     PlcTask Outputs/GVL_iXlinker.EtherCAT_Master_BKCUCX.TcTerminals210_EK1100_1.TcTerminals210_1BK1250.A_0213_KL_2545_2_Ch_PWM_Amplifier_50V_3_5_A.Channel_2.Data_Out <-> Channel 2/Data Out
//   PLC/PLC Instance <-> EtherCAT Master BKCUCX/TcTerminals210_EK1100_1/TcTerminals210_1BK1250/A_0214(KL 2552, 2 Ch. DC Amplifier (50V, 3.5 A))
//     PlcTask Inputs/GVL_iXlinker.EtherCAT_Master_BKCUCX.TcTerminals210_EK1100_1.TcTerminals210_1BK1250.A_0214_KL_2552_2_Ch_DC_Amplifier_50V_3_5_A.Channel_1.State <-> Channel 1/State
//     PlcTask Inputs/GVL_iXlinker.EtherCAT_Master_BKCUCX.TcTerminals210_EK1100_1.TcTerminals210_1BK1250.A_0214_KL_2552_2_Ch_DC_Amplifier_50V_3_5_A.Channel_2.State <-> Channel 2/State
//     PlcTask Inputs/GVL_iXlinker.EtherCAT_Master_BKCUCX.TcTerminals210_EK1100_1.TcTerminals210_1BK1250.A_0214_KL_2552_2_Ch_DC_Amplifier_50V_3_5_A.Channel_1.Data_In <-> Channel 1/Data In
//     PlcTask Inputs/GVL_iXlinker.EtherCAT_Master_BKCUCX.TcTerminals210_EK1100_1.TcTerminals210_1BK1250.A_0214_KL_2552_2_Ch_DC_Amplifier_50V_3_5_A.Channel_2.Data_In <-> Channel 2/Data In
//     PlcTask Outputs/GVL_iXlinker.EtherCAT_Master_BKCUCX.TcTerminals210_EK1100_1.TcTerminals210_1BK1250.A_0214_KL_2552_2_Ch_DC_Amplifier_50V_3_5_A.Channel_1.Ctrl <-> Channel 1/Ctrl
//     PlcTask Outputs/GVL_iXlinker.EtherCAT_Master_BKCUCX.TcTerminals210_EK1100_1.TcTerminals210_1BK1250.A_0214_KL_2552_2_Ch_DC_Amplifier_50V_3_5_A.Channel_2.Ctrl <-> Channel 2/Ctrl
//     PlcTask Outputs/GVL_iXlinker.EtherCAT_Master_BKCUCX.TcTerminals210_EK1100_1.TcTerminals210_1BK1250.A_0214_KL_2552_2_Ch_DC_Amplifier_50V_3_5_A.Channel_1.Data_Out <-> Channel 1/Data Out
//     PlcTask Outputs/GVL_iXlinker.EtherCAT_Master_BKCUCX.TcTerminals210_EK1100_1.TcTerminals210_1BK1250.A_0214_KL_2552_2_Ch_DC_Amplifier_50V_3_5_A.Channel_2.Data_Out <-> Channel 2/Data Out
//   PLC/PLC Instance <-> EtherCAT Master BKCUCX/TcTerminals210_EK1100_1/TcTerminals210_1BK1250/A_0215(KL 2602, 2 Ch. Output Relay (230V AC/ 30V DC))
//     PlcTask Outputs/GVL_iXlinker.EtherCAT_Master_BKCUCX.TcTerminals210_EK1100_1.TcTerminals210_1BK1250.A_0215_KL_2602_2_Ch_Output_Relay_230V_AC_30V_DC.Channel_1.Output <-> Channel 1/Output
//     PlcTask Outputs/GVL_iXlinker.EtherCAT_Master_BKCUCX.TcTerminals210_EK1100_1.TcTerminals210_1BK1250.A_0215_KL_2602_2_Ch_Output_Relay_230V_AC_30V_DC.Channel_2.Output <-> Channel 2/Output
//   PLC/PLC Instance <-> EtherCAT Master BKCUCX/TcTerminals210_EK1100_1/TcTerminals210_1BK1250/A_0216(KL 2602-0010, 2 Ch. Output Relay + ZCD (230V AC/ 30V DC))
//     PlcTask Outputs/GVL_iXlinker.EtherCAT_Master_BKCUCX.TcTerminals210_EK1100_1.TcTerminals210_1BK1250.A_0216_KL_2602_0010_2_Ch_Output_Relay_ZCD_230V_AC_30V_DC.Channel_1.Output <-> Channel 1/Output
//     PlcTask Outputs/GVL_iXlinker.EtherCAT_Master_BKCUCX.TcTerminals210_EK1100_1.TcTerminals210_1BK1250.A_0216_KL_2602_0010_2_Ch_Output_Relay_ZCD_230V_AC_30V_DC.Channel_2.Output <-> Channel 2/Output
//   PLC/PLC Instance <-> EtherCAT Master BKCUCX/TcTerminals210_EK1100_1/TcTerminals210_1BK1250/A_0217(KL 2612, 2 Ch. Output Relay (125V AC/ 30V DC))
//     PlcTask Outputs/GVL_iXlinker.EtherCAT_Master_BKCUCX.TcTerminals210_EK1100_1.TcTerminals210_1BK1250.A_0217_KL_2612_2_Ch_Output_Relay_125V_AC_30V_DC.Channel_1.Output <-> Channel 1/Output
//     PlcTask Outputs/GVL_iXlinker.EtherCAT_Master_BKCUCX.TcTerminals210_EK1100_1.TcTerminals210_1BK1250.A_0217_KL_2612_2_Ch_Output_Relay_125V_AC_30V_DC.Channel_2.Output <-> Channel 2/Output
//   PLC/PLC Instance <-> EtherCAT Master BKCUCX/TcTerminals210_EK1100_1/TcTerminals210_1BK1250/A_0218(KL 2622, 2 Ch. Output Relay (230V AC/ 30V DC))
//     PlcTask Outputs/GVL_iXlinker.EtherCAT_Master_BKCUCX.TcTerminals210_EK1100_1.TcTerminals210_1BK1250.A_0218_KL_2622_2_Ch_Output_Relay_230V_AC_30V_DC.Channel_1.Output <-> Channel 1/Output
//     PlcTask Outputs/GVL_iXlinker.EtherCAT_Master_BKCUCX.TcTerminals210_EK1100_1.TcTerminals210_1BK1250.A_0218_KL_2622_2_Ch_Output_Relay_230V_AC_30V_DC.Channel_2.Output <-> Channel 2/Output
//   PLC/PLC Instance <-> EtherCAT Master BKCUCX/TcTerminals210_EK1100_1/TcTerminals210_1BK1250/A_0219(KL 2622-0010, 2 Ch. Output Relay + ZCD (230V AC/ 30V DC))
//     PlcTask Outputs/GVL_iXlinker.EtherCAT_Master_BKCUCX.TcTerminals210_EK1100_1.TcTerminals210_1BK1250.A_0219_KL_2622_0010_2_Ch_Output_Relay_ZCD_230V_AC_30V_DC.Channel_1.Output <-> Channel 1/Output
//     PlcTask Outputs/GVL_iXlinker.EtherCAT_Master_BKCUCX.TcTerminals210_EK1100_1.TcTerminals210_1BK1250.A_0219_KL_2622_0010_2_Ch_Output_Relay_ZCD_230V_AC_30V_DC.Channel_2.Output <-> Channel 2/Output
//   PLC/PLC Instance <-> EtherCAT Master BKCUCX/TcTerminals210_EK1100_1/TcTerminals210_1BK1250/A_0220(KL 2631, 1 Ch. Power Output Relay (400V AC/ 3A))
//     PlcTask Outputs/GVL_iXlinker.EtherCAT_Master_BKCUCX.TcTerminals210_EK1100_1.TcTerminals210_1BK1250.A_0220_KL_2631_1_Ch_Power_Output_Relay_400V_AC_3A.Channel_1.Output <-> Channel 1/Output
//   PLC/PLC Instance <-> EtherCAT Master BKCUCX/TcTerminals210_EK1100_1/TcTerminals210_1BK1250/A_0221(KL 2634, 4 Ch. Power Output Relay (250 V AC/30 V DC))
//     PlcTask Outputs/GVL_iXlinker.EtherCAT_Master_BKCUCX.TcTerminals210_EK1100_1.TcTerminals210_1BK1250.A_0221_KL_2634_4_Ch_Power_Output_Relay_250_V_AC_30_V_DC.Channel_1.Output <-> Channel 1/Output
//     PlcTask Outputs/GVL_iXlinker.EtherCAT_Master_BKCUCX.TcTerminals210_EK1100_1.TcTerminals210_1BK1250.A_0221_KL_2634_4_Ch_Power_Output_Relay_250_V_AC_30_V_DC.Channel_2.Output <-> Channel 2/Output
//     PlcTask Outputs/GVL_iXlinker.EtherCAT_Master_BKCUCX.TcTerminals210_EK1100_1.TcTerminals210_1BK1250.A_0221_KL_2634_4_Ch_Power_Output_Relay_250_V_AC_30_V_DC.Channel_3.Output <-> Channel 3/Output
//     PlcTask Outputs/GVL_iXlinker.EtherCAT_Master_BKCUCX.TcTerminals210_EK1100_1.TcTerminals210_1BK1250.A_0221_KL_2634_4_Ch_Power_Output_Relay_250_V_AC_30_V_DC.Channel_4.Output <-> Channel 4/Output
//   PLC/PLC Instance <-> EtherCAT Master BKCUCX/TcTerminals210_EK1100_1/TcTerminals210_1BK1250/A_0222(KL 2641, 1 Ch. Power Output Relay (230V AC/ 16A))
//     PlcTask Inputs/GVL_iXlinker.EtherCAT_Master_BKCUCX.TcTerminals210_EK1100_1.TcTerminals210_1BK1250.A_0222_KL_2641_1_Ch_Power_Output_Relay_230V_AC_16A.Channel_1.State <-> Channel 1/State
//     PlcTask Outputs/GVL_iXlinker.EtherCAT_Master_BKCUCX.TcTerminals210_EK1100_1.TcTerminals210_1BK1250.A_0222_KL_2641_1_Ch_Power_Output_Relay_230V_AC_16A.Channel_1.Output <-> Channel 1/Output
//   PLC/PLC Instance <-> EtherCAT Master BKCUCX/TcTerminals210_EK1100_1/TcTerminals210_1BK1250/A_0223(KL 2641, 1 Ch. Power Output Relay (230V AC/ 16A))
//     PlcTask Inputs/GVL_iXlinker.EtherCAT_Master_BKCUCX.TcTerminals210_EK1100_1.TcTerminals210_1BK1250.A_0223_KL_2641_1_Ch_Power_Output_Relay_230V_AC_16A.Channel_1.Manual_State <-> Channel 1/Manual State
//     PlcTask Inputs/GVL_iXlinker.EtherCAT_Master_BKCUCX.TcTerminals210_EK1100_1.TcTerminals210_1BK1250.A_0223_KL_2641_1_Ch_Power_Output_Relay_230V_AC_16A.Channel_1.Reserved <-> Channel 1/Reserved
//     PlcTask Outputs/GVL_iXlinker.EtherCAT_Master_BKCUCX.TcTerminals210_EK1100_1.TcTerminals210_1BK1250.A_0223_KL_2641_1_Ch_Power_Output_Relay_230V_AC_16A.Channel_1.Output <-> Channel 1/Output
//   PLC/PLC Instance <-> EtherCAT Master BKCUCX/TcTerminals210_EK1100_1/TcTerminals210_1BK1250/A_0224(KL 2652, 2 Ch. Power Output Relay (230V AC/ 1A))
//     PlcTask Outputs/GVL_iXlinker.EtherCAT_Master_BKCUCX.TcTerminals210_EK1100_1.TcTerminals210_1BK1250.A_0224_KL_2652_2_Ch_Power_Output_Relay_230V_AC_1A.Channel_1.Output <-> Channel 1/Output
//     PlcTask Outputs/GVL_iXlinker.EtherCAT_Master_BKCUCX.TcTerminals210_EK1100_1.TcTerminals210_1BK1250.A_0224_KL_2652_2_Ch_Power_Output_Relay_230V_AC_1A.Channel_2.Output <-> Channel 2/Output
//   PLC/PLC Instance <-> EtherCAT Master BKCUCX/TcTerminals210_EK1100_1/TcTerminals210_1BK1250/A_0225(KL 2692, Cycle Monitoring Terminal)
//     PlcTask Inputs/GVL_iXlinker.EtherCAT_Master_BKCUCX.TcTerminals210_EK1100_1.TcTerminals210_1BK1250.A_0225_KL_2692_Cycle_Monitoring_Terminal.Channel_1.State <-> Channel 1/State
//     PlcTask Inputs/GVL_iXlinker.EtherCAT_Master_BKCUCX.TcTerminals210_EK1100_1.TcTerminals210_1BK1250.A_0225_KL_2692_Cycle_Monitoring_Terminal.Channel_1.Data_In <-> Channel 1/Data In
//     PlcTask Outputs/GVL_iXlinker.EtherCAT_Master_BKCUCX.TcTerminals210_EK1100_1.TcTerminals210_1BK1250.A_0225_KL_2692_Cycle_Monitoring_Terminal.Channel_1.Ctrl <-> Channel 1/Ctrl
//     PlcTask Outputs/GVL_iXlinker.EtherCAT_Master_BKCUCX.TcTerminals210_EK1100_1.TcTerminals210_1BK1250.A_0225_KL_2692_Cycle_Monitoring_Terminal.Channel_1.Data_Out <-> Channel 1/Data Out
//   PLC/PLC Instance <-> EtherCAT Master BKCUCX/TcTerminals210_EK1100_1/TcTerminals210_1BK1250/A_0226(KL 2701, 1 Ch.  Solid State Load Relay (230V AC/ 3A))
//     PlcTask Outputs/GVL_iXlinker.EtherCAT_Master_BKCUCX.TcTerminals210_EK1100_1.TcTerminals210_1BK1250.A_0226_KL_2701_1_Ch_Solid_State_Load_Relay_230V_AC_3A.Channel_1.Output <-> Channel 1/Output
//   PLC/PLC Instance <-> EtherCAT Master BKCUCX/TcTerminals210_EK1100_1/TcTerminals210_1BK1250/A_0227(KL 2702, 2 Ch. Output Solid State Relay (230V AC/DC, 0.3A))
//     PlcTask Outputs/GVL_iXlinker.EtherCAT_Master_BKCUCX.TcTerminals210_EK1100_1.TcTerminals210_1BK1250.A_0227_KL_2702_2_Ch_Output_Solid_State_Relay_230V_AC_DC_0_3A.Channel_1.Output <-> Channel 1/Output
//     PlcTask Outputs/GVL_iXlinker.EtherCAT_Master_BKCUCX.TcTerminals210_EK1100_1.TcTerminals210_1BK1250.A_0227_KL_2702_2_Ch_Output_Solid_State_Relay_230V_AC_DC_0_3A.Channel_2.Output <-> Channel 2/Output
//   PLC/PLC Instance <-> EtherCAT Master BKCUCX/TcTerminals210_EK1100_1/TcTerminals210_1BK1250/A_0228(KL 2702-0002, 2 Ch. Output Solid State Relay (230V AC/DC, 2A, mutually locked))
//     PlcTask Outputs/GVL_iXlinker.EtherCAT_Master_BKCUCX.TcTerminals210_EK1100_1.TcTerminals210_1BK1250.A_0228_KL_2702_0002_2_Ch_Output_Solid_State_Relay_230V_AC_DC_2A_mutually_locked.Channel_1.Output <-> Channel 1/Output
//     PlcTask Outputs/GVL_iXlinker.EtherCAT_Master_BKCUCX.TcTerminals210_EK1100_1.TcTerminals210_1BK1250.A_0228_KL_2702_0002_2_Ch_Output_Solid_State_Relay_230V_AC_DC_2A_mutually_locked.Channel_2.Output <-> Channel 2/Output
//   PLC/PLC Instance <-> EtherCAT Master BKCUCX/TcTerminals210_EK1100_1/TcTerminals210_1BK1250/A_0229(KL 2702-0020, 2 Ch. Output Solid State Relay (230V AC/DC, 1.5A))
//     PlcTask Outputs/GVL_iXlinker.EtherCAT_Master_BKCUCX.TcTerminals210_EK1100_1.TcTerminals210_1BK1250.A_0229_KL_2702_0020_2_Ch_Output_Solid_State_Relay_230V_AC_DC_1_5A.Channel_1.Output <-> Channel 1/Output
//     PlcTask Outputs/GVL_iXlinker.EtherCAT_Master_BKCUCX.TcTerminals210_EK1100_1.TcTerminals210_1BK1250.A_0229_KL_2702_0020_2_Ch_Output_Solid_State_Relay_230V_AC_DC_1_5A.Channel_2.Output <-> Channel 2/Output
//   PLC/PLC Instance <-> EtherCAT Master BKCUCX/TcTerminals210_EK1100_1/TcTerminals210_1BK1250/A_0230(KL 2712, 2 Ch. Triac Output (12-230V AC, 0.5A))
//     PlcTask Outputs/GVL_iXlinker.EtherCAT_Master_BKCUCX.TcTerminals210_EK1100_1.TcTerminals210_1BK1250.A_0230_KL_2712_2_Ch_Triac_Output_12_230V_AC_0_5A.Channel_1.Output <-> Channel 1/Output
//     PlcTask Outputs/GVL_iXlinker.EtherCAT_Master_BKCUCX.TcTerminals210_EK1100_1.TcTerminals210_1BK1250.A_0230_KL_2712_2_Ch_Triac_Output_12_230V_AC_0_5A.Channel_2.Output <-> Channel 2/Output
//   PLC/PLC Instance <-> EtherCAT Master BKCUCX/TcTerminals210_EK1100_1/TcTerminals210_1BK1250/A_0231(KL 2722, 2 Ch. Triac Output (12-230V AC, 0.01-1A))
//     PlcTask Outputs/GVL_iXlinker.EtherCAT_Master_BKCUCX.TcTerminals210_EK1100_1.TcTerminals210_1BK1250.A_0231_KL_2722_2_Ch_Triac_Output_12_230V_AC_0_01_1A.Channel_1.Output <-> Channel 1/Output
//     PlcTask Outputs/GVL_iXlinker.EtherCAT_Master_BKCUCX.TcTerminals210_EK1100_1.TcTerminals210_1BK1250.A_0231_KL_2722_2_Ch_Triac_Output_12_230V_AC_0_01_1A.Channel_2.Output <-> Channel 2/Output
//   PLC/PLC Instance <-> EtherCAT Master BKCUCX/TcTerminals210_EK1100_1/TcTerminals210_1BK1250/A_0232(KL 2732, 2 Ch. Triac Output (12-230V AC, 0.01-1A, no power contacts))
//     PlcTask Outputs/GVL_iXlinker.EtherCAT_Master_BKCUCX.TcTerminals210_EK1100_1.TcTerminals210_1BK1250.A_0232_KL_2732_2_Ch_Triac_Output_12_230V_AC_0_01_1A_no_power_contacts.Channel_1.Output <-> Channel 1/Output
//     PlcTask Outputs/GVL_iXlinker.EtherCAT_Master_BKCUCX.TcTerminals210_EK1100_1.TcTerminals210_1BK1250.A_0232_KL_2732_2_Ch_Triac_Output_12_230V_AC_0_01_1A_no_power_contacts.Channel_2.Output <-> Channel 2/Output
//   PLC/PLC Instance <-> EtherCAT Master BKCUCX/TcTerminals210_EK1100_1/TcTerminals210_1BK1250/A_0233(KL 2744, 4 Ch. Output Solid State Relay (230V AC/DC, 1.5A))
//     PlcTask Outputs/GVL_iXlinker.EtherCAT_Master_BKCUCX.TcTerminals210_EK1100_1.TcTerminals210_1BK1250.A_0233_KL_2744_4_Ch_Output_Solid_State_Relay_230V_AC_DC_1_5A.Channel_1.Output <-> Channel 1/Output
//     PlcTask Outputs/GVL_iXlinker.EtherCAT_Master_BKCUCX.TcTerminals210_EK1100_1.TcTerminals210_1BK1250.A_0233_KL_2744_4_Ch_Output_Solid_State_Relay_230V_AC_DC_1_5A.Channel_2.Output <-> Channel 2/Output
//     PlcTask Outputs/GVL_iXlinker.EtherCAT_Master_BKCUCX.TcTerminals210_EK1100_1.TcTerminals210_1BK1250.A_0233_KL_2744_4_Ch_Output_Solid_State_Relay_230V_AC_DC_1_5A.Channel_3.Output <-> Channel 3/Output
//     PlcTask Outputs/GVL_iXlinker.EtherCAT_Master_BKCUCX.TcTerminals210_EK1100_1.TcTerminals210_1BK1250.A_0233_KL_2744_4_Ch_Output_Solid_State_Relay_230V_AC_DC_1_5A.Channel_4.Output <-> Channel 4/Output
//   PLC/PLC Instance <-> EtherCAT Master BKCUCX/TcTerminals210_EK1100_1/TcTerminals210_1BK1250/A_0234(KL 2751, 1 Ch. Universal Dimmer (230V AC, 300VA))
//     PlcTask Inputs/GVL_iXlinker.EtherCAT_Master_BKCUCX.TcTerminals210_EK1100_1.TcTerminals210_1BK1250.A_0234_KL_2751_1_Ch_Universal_Dimmer_230V_AC_300VA.Channel_1.State <-> Channel 1/State
//     PlcTask Inputs/GVL_iXlinker.EtherCAT_Master_BKCUCX.TcTerminals210_EK1100_1.TcTerminals210_1BK1250.A_0234_KL_2751_1_Ch_Universal_Dimmer_230V_AC_300VA.Channel_1.Data_In <-> Channel 1/Data In
//     PlcTask Outputs/GVL_iXlinker.EtherCAT_Master_BKCUCX.TcTerminals210_EK1100_1.TcTerminals210_1BK1250.A_0234_KL_2751_1_Ch_Universal_Dimmer_230V_AC_300VA.Channel_1.Ctrl <-> Channel 1/Ctrl
//     PlcTask Outputs/GVL_iXlinker.EtherCAT_Master_BKCUCX.TcTerminals210_EK1100_1.TcTerminals210_1BK1250.A_0234_KL_2751_1_Ch_Universal_Dimmer_230V_AC_300VA.Channel_1.Data_Out <-> Channel 1/Data Out
//   PLC/PLC Instance <-> EtherCAT Master BKCUCX/TcTerminals210_EK1100_1/TcTerminals210_1BK1250/A_0236(KL 2751-1200, 1 Ch. Universal Dimmer (120V AC, 300VA))
//     PlcTask Inputs/GVL_iXlinker.EtherCAT_Master_BKCUCX.TcTerminals210_EK1100_1.TcTerminals210_1BK1250.A_0236_KL_2751_1200_1_Ch_Universal_Dimmer_120V_AC_300VA.Channel_1.State <-> Channel 1/State
//     PlcTask Inputs/GVL_iXlinker.EtherCAT_Master_BKCUCX.TcTerminals210_EK1100_1.TcTerminals210_1BK1250.A_0236_KL_2751_1200_1_Ch_Universal_Dimmer_120V_AC_300VA.Channel_1.Data_In <-> Channel 1/Data In
//     PlcTask Outputs/GVL_iXlinker.EtherCAT_Master_BKCUCX.TcTerminals210_EK1100_1.TcTerminals210_1BK1250.A_0236_KL_2751_1200_1_Ch_Universal_Dimmer_120V_AC_300VA.Channel_1.Ctrl <-> Channel 1/Ctrl
//     PlcTask Outputs/GVL_iXlinker.EtherCAT_Master_BKCUCX.TcTerminals210_EK1100_1.TcTerminals210_1BK1250.A_0236_KL_2751_1200_1_Ch_Universal_Dimmer_120V_AC_300VA.Channel_1.Data_Out <-> Channel 1/Data Out
//   PLC/PLC Instance <-> EtherCAT Master BKCUCX/TcTerminals210_EK1100_1/TcTerminals210_1BK1250/A_0238(KL 2761, 1 Ch. Universal Dimmer (230V AC, 600VA))
//     PlcTask Inputs/GVL_iXlinker.EtherCAT_Master_BKCUCX.TcTerminals210_EK1100_1.TcTerminals210_1BK1250.A_0238_KL_2761_1_Ch_Universal_Dimmer_230V_AC_600VA.Channel_1.State <-> Channel 1/State
//     PlcTask Inputs/GVL_iXlinker.EtherCAT_Master_BKCUCX.TcTerminals210_EK1100_1.TcTerminals210_1BK1250.A_0238_KL_2761_1_Ch_Universal_Dimmer_230V_AC_600VA.Channel_1.Data_In <-> Channel 1/Data In
//     PlcTask Outputs/GVL_iXlinker.EtherCAT_Master_BKCUCX.TcTerminals210_EK1100_1.TcTerminals210_1BK1250.A_0238_KL_2761_1_Ch_Universal_Dimmer_230V_AC_600VA.Channel_1.Ctrl <-> Channel 1/Ctrl
//     PlcTask Outputs/GVL_iXlinker.EtherCAT_Master_BKCUCX.TcTerminals210_EK1100_1.TcTerminals210_1BK1250.A_0238_KL_2761_1_Ch_Universal_Dimmer_230V_AC_600VA.Channel_1.Data_Out <-> Channel 1/Data Out
//   PLC/PLC Instance <-> EtherCAT Master BKCUCX/TcTerminals210_EK1100_1/TcTerminals210_1BK1250/A_0240(KL 2784, 4 Ch. Output (24V AC/DC, 2A, short-circut-proof))
//     PlcTask Outputs/GVL_iXlinker.EtherCAT_Master_BKCUCX.TcTerminals210_EK1100_1.TcTerminals210_1BK1250.A_0240_KL_2784_4_Ch_Output_24V_AC_DC_2A_short_circut_proof.Channel_1.Output <-> Channel 1/Output
//     PlcTask Outputs/GVL_iXlinker.EtherCAT_Master_BKCUCX.TcTerminals210_EK1100_1.TcTerminals210_1BK1250.A_0240_KL_2784_4_Ch_Output_24V_AC_DC_2A_short_circut_proof.Channel_2.Output <-> Channel 2/Output
//     PlcTask Outputs/GVL_iXlinker.EtherCAT_Master_BKCUCX.TcTerminals210_EK1100_1.TcTerminals210_1BK1250.A_0240_KL_2784_4_Ch_Output_24V_AC_DC_2A_short_circut_proof.Channel_3.Output <-> Channel 3/Output
//     PlcTask Outputs/GVL_iXlinker.EtherCAT_Master_BKCUCX.TcTerminals210_EK1100_1.TcTerminals210_1BK1250.A_0240_KL_2784_4_Ch_Output_24V_AC_DC_2A_short_circut_proof.Channel_4.Output <-> Channel 4/Output
//   PLC/PLC Instance <-> EtherCAT Master BKCUCX/TcTerminals210_EK1100_1/TcTerminals210_1BK1250/A_0241(KL 2791, 1 Ch. Speed Controller (230V AC, 100 VA))
//     PlcTask Inputs/GVL_iXlinker.EtherCAT_Master_BKCUCX.TcTerminals210_EK1100_1.TcTerminals210_1BK1250.A_0241_KL_2791_1_Ch_Speed_Controller_230V_AC_100_VA.Channel_1.State <-> Channel 1/State
//     PlcTask Inputs/GVL_iXlinker.EtherCAT_Master_BKCUCX.TcTerminals210_EK1100_1.TcTerminals210_1BK1250.A_0241_KL_2791_1_Ch_Speed_Controller_230V_AC_100_VA.Channel_1.Data_In <-> Channel 1/Data In
//     PlcTask Outputs/GVL_iXlinker.EtherCAT_Master_BKCUCX.TcTerminals210_EK1100_1.TcTerminals210_1BK1250.A_0241_KL_2791_1_Ch_Speed_Controller_230V_AC_100_VA.Channel_1.Ctrl <-> Channel 1/Ctrl
//     PlcTask Outputs/GVL_iXlinker.EtherCAT_Master_BKCUCX.TcTerminals210_EK1100_1.TcTerminals210_1BK1250.A_0241_KL_2791_1_Ch_Speed_Controller_230V_AC_100_VA.Channel_1.Data_Out <-> Channel 1/Data Out
//   PLC/PLC Instance <-> EtherCAT Master BKCUCX/TcTerminals210_EK1100_1/TcTerminals210_1BK1250/A_0243(KL 2791-1200, 1 Ch. Speed Controller (120V AC, 100 VA))
//     PlcTask Inputs/GVL_iXlinker.EtherCAT_Master_BKCUCX.TcTerminals210_EK1100_1.TcTerminals210_1BK1250.A_0243_KL_2791_1200_1_Ch_Speed_Controller_120V_AC_100_VA.Channel_1.State <-> Channel 1/State
//     PlcTask Inputs/GVL_iXlinker.EtherCAT_Master_BKCUCX.TcTerminals210_EK1100_1.TcTerminals210_1BK1250.A_0243_KL_2791_1200_1_Ch_Speed_Controller_120V_AC_100_VA.Channel_1.Data_In <-> Channel 1/Data In
//     PlcTask Outputs/GVL_iXlinker.EtherCAT_Master_BKCUCX.TcTerminals210_EK1100_1.TcTerminals210_1BK1250.A_0243_KL_2791_1200_1_Ch_Speed_Controller_120V_AC_100_VA.Channel_1.Ctrl <-> Channel 1/Ctrl
//     PlcTask Outputs/GVL_iXlinker.EtherCAT_Master_BKCUCX.TcTerminals210_EK1100_1.TcTerminals210_1BK1250.A_0243_KL_2791_1200_1_Ch_Speed_Controller_120V_AC_100_VA.Channel_1.Data_Out <-> Channel 1/Data Out
//   PLC/PLC Instance <-> EtherCAT Master BKCUCX/TcTerminals210_EK1100_1/TcTerminals210_1BK1250/A_0245(KL 2794, 4 Ch. Output (24V AC/DC, 2A, potential-free, short-circut-proof))
//     PlcTask Outputs/GVL_iXlinker.EtherCAT_Master_BKCUCX.TcTerminals210_EK1100_1.TcTerminals210_1BK1250.A_0245_KL_2794_4_Ch_Output_24V_AC_DC_2A_potential_free_short_circut_proof.Channel_1.Output <-> Channel 1/Output
//     PlcTask Outputs/GVL_iXlinker.EtherCAT_Master_BKCUCX.TcTerminals210_EK1100_1.TcTerminals210_1BK1250.A_0245_KL_2794_4_Ch_Output_24V_AC_DC_2A_potential_free_short_circut_proof.Channel_2.Output <-> Channel 2/Output
//     PlcTask Outputs/GVL_iXlinker.EtherCAT_Master_BKCUCX.TcTerminals210_EK1100_1.TcTerminals210_1BK1250.A_0245_KL_2794_4_Ch_Output_24V_AC_DC_2A_potential_free_short_circut_proof.Channel_3.Output <-> Channel 3/Output
//     PlcTask Outputs/GVL_iXlinker.EtherCAT_Master_BKCUCX.TcTerminals210_EK1100_1.TcTerminals210_1BK1250.A_0245_KL_2794_4_Ch_Output_24V_AC_DC_2A_potential_free_short_circut_proof.Channel_4.Output <-> Channel 4/Output
//   PLC/PLC Instance <-> EtherCAT Master BKCUCX/TcTerminals210_EK1100_1/TcTerminals210_1BK1250/A_0246(KL 2798, 8 Ch. Output (24V AC/DC, 2A, potential-free, short-circut-proof))
//     PlcTask Outputs/GVL_iXlinker.EtherCAT_Master_BKCUCX.TcTerminals210_EK1100_1.TcTerminals210_1BK1250.A_0246_KL_2798_8_Ch_Output_24V_AC_DC_2A_potential_free_short_circut_proof.Channel_1.Output <-> Channel 1/Output
//     PlcTask Outputs/GVL_iXlinker.EtherCAT_Master_BKCUCX.TcTerminals210_EK1100_1.TcTerminals210_1BK1250.A_0246_KL_2798_8_Ch_Output_24V_AC_DC_2A_potential_free_short_circut_proof.Channel_2.Output <-> Channel 2/Output
//     PlcTask Outputs/GVL_iXlinker.EtherCAT_Master_BKCUCX.TcTerminals210_EK1100_1.TcTerminals210_1BK1250.A_0246_KL_2798_8_Ch_Output_24V_AC_DC_2A_potential_free_short_circut_proof.Channel_3.Output <-> Channel 3/Output
//     PlcTask Outputs/GVL_iXlinker.EtherCAT_Master_BKCUCX.TcTerminals210_EK1100_1.TcTerminals210_1BK1250.A_0246_KL_2798_8_Ch_Output_24V_AC_DC_2A_potential_free_short_circut_proof.Channel_4.Output <-> Channel 4/Output
//     PlcTask Outputs/GVL_iXlinker.EtherCAT_Master_BKCUCX.TcTerminals210_EK1100_1.TcTerminals210_1BK1250.A_0246_KL_2798_8_Ch_Output_24V_AC_DC_2A_potential_free_short_circut_proof.Channel_5.Output <-> Channel 5/Output
//     PlcTask Outputs/GVL_iXlinker.EtherCAT_Master_BKCUCX.TcTerminals210_EK1100_1.TcTerminals210_1BK1250.A_0246_KL_2798_8_Ch_Output_24V_AC_DC_2A_potential_free_short_circut_proof.Channel_6.Output <-> Channel 6/Output
//     PlcTask Outputs/GVL_iXlinker.EtherCAT_Master_BKCUCX.TcTerminals210_EK1100_1.TcTerminals210_1BK1250.A_0246_KL_2798_8_Ch_Output_24V_AC_DC_2A_potential_free_short_circut_proof.Channel_7.Output <-> Channel 7/Output
//     PlcTask Outputs/GVL_iXlinker.EtherCAT_Master_BKCUCX.TcTerminals210_EK1100_1.TcTerminals210_1BK1250.A_0246_KL_2798_8_Ch_Output_24V_AC_DC_2A_potential_free_short_circut_proof.Channel_8.Output <-> Channel 8/Output
//   PLC/PLC Instance <-> EtherCAT Master BKCUCX/TcTerminals210_EK1100_1/TcTerminals210_1BK1250/A_0247(KL 2808, 8 Ch. Output with Protection (24V, 0.5 A, 2 wire))
//     PlcTask Outputs/GVL_iXlinker.EtherCAT_Master_BKCUCX.TcTerminals210_EK1100_1.TcTerminals210_1BK1250.A_0247_KL_2808_8_Ch_Output_with_Protection_24V_0_5_A_2_wire.Channel_1.Output <-> Channel 1/Output
//     PlcTask Outputs/GVL_iXlinker.EtherCAT_Master_BKCUCX.TcTerminals210_EK1100_1.TcTerminals210_1BK1250.A_0247_KL_2808_8_Ch_Output_with_Protection_24V_0_5_A_2_wire.Channel_2.Output <-> Channel 2/Output
//     PlcTask Outputs/GVL_iXlinker.EtherCAT_Master_BKCUCX.TcTerminals210_EK1100_1.TcTerminals210_1BK1250.A_0247_KL_2808_8_Ch_Output_with_Protection_24V_0_5_A_2_wire.Channel_3.Output <-> Channel 3/Output
//     PlcTask Outputs/GVL_iXlinker.EtherCAT_Master_BKCUCX.TcTerminals210_EK1100_1.TcTerminals210_1BK1250.A_0247_KL_2808_8_Ch_Output_with_Protection_24V_0_5_A_2_wire.Channel_4.Output <-> Channel 4/Output
//     PlcTask Outputs/GVL_iXlinker.EtherCAT_Master_BKCUCX.TcTerminals210_EK1100_1.TcTerminals210_1BK1250.A_0247_KL_2808_8_Ch_Output_with_Protection_24V_0_5_A_2_wire.Channel_5.Output <-> Channel 5/Output
//     PlcTask Outputs/GVL_iXlinker.EtherCAT_Master_BKCUCX.TcTerminals210_EK1100_1.TcTerminals210_1BK1250.A_0247_KL_2808_8_Ch_Output_with_Protection_24V_0_5_A_2_wire.Channel_6.Output <-> Channel 6/Output
//     PlcTask Outputs/GVL_iXlinker.EtherCAT_Master_BKCUCX.TcTerminals210_EK1100_1.TcTerminals210_1BK1250.A_0247_KL_2808_8_Ch_Output_with_Protection_24V_0_5_A_2_wire.Channel_7.Output <-> Channel 7/Output
//     PlcTask Outputs/GVL_iXlinker.EtherCAT_Master_BKCUCX.TcTerminals210_EK1100_1.TcTerminals210_1BK1250.A_0247_KL_2808_8_Ch_Output_with_Protection_24V_0_5_A_2_wire.Channel_8.Output <-> Channel 8/Output
//   PLC/PLC Instance <-> EtherCAT Master BKCUCX/TcTerminals210_EK1100_1/TcTerminals210_1BK1250/A_0248(KL 2819, 16 Ch. Output (24V, 0.5 A) with Diagnostic complex)
//     PlcTask Inputs/GVL_iXlinker.EtherCAT_Master_BKCUCX.TcTerminals210_EK1100_1.TcTerminals210_1BK1250.A_0248_KL_2819_16_Ch_Output_24V_0_5_A_with_Diagnostic_complex.Channel_1.Status <-> Channel 1/Status
//     PlcTask Inputs/GVL_iXlinker.EtherCAT_Master_BKCUCX.TcTerminals210_EK1100_1.TcTerminals210_1BK1250.A_0248_KL_2819_16_Ch_Output_24V_0_5_A_with_Diagnostic_complex.Channel_1.Diag <-> Channel 1/Diag
//     PlcTask Outputs/GVL_iXlinker.EtherCAT_Master_BKCUCX.TcTerminals210_EK1100_1.TcTerminals210_1BK1250.A_0248_KL_2819_16_Ch_Output_24V_0_5_A_with_Diagnostic_complex.Channel_1.Ctrl <-> Channel 1/Ctrl
//     PlcTask Outputs/GVL_iXlinker.EtherCAT_Master_BKCUCX.TcTerminals210_EK1100_1.TcTerminals210_1BK1250.A_0248_KL_2819_16_Ch_Output_24V_0_5_A_with_Diagnostic_complex.Channel_1.Output <-> Channel 1/Output
//   PLC/PLC Instance <-> EtherCAT Master BKCUCX/TcTerminals210_EK1100_1/TcTerminals210_1BK1250/A_0250(KL 2828, 8 Ch. Output with Protection (24V, 2.0 A, 2 wire))
//     PlcTask Outputs/GVL_iXlinker.EtherCAT_Master_BKCUCX.TcTerminals210_EK1100_1.TcTerminals210_1BK1250.A_0250_KL_2828_8_Ch_Output_with_Protection_24V_2_0_A_2_wire.Channel_1.Output <-> Channel 1/Output
//     PlcTask Outputs/GVL_iXlinker.EtherCAT_Master_BKCUCX.TcTerminals210_EK1100_1.TcTerminals210_1BK1250.A_0250_KL_2828_8_Ch_Output_with_Protection_24V_2_0_A_2_wire.Channel_2.Output <-> Channel 2/Output
//     PlcTask Outputs/GVL_iXlinker.EtherCAT_Master_BKCUCX.TcTerminals210_EK1100_1.TcTerminals210_1BK1250.A_0250_KL_2828_8_Ch_Output_with_Protection_24V_2_0_A_2_wire.Channel_3.Output <-> Channel 3/Output
//     PlcTask Outputs/GVL_iXlinker.EtherCAT_Master_BKCUCX.TcTerminals210_EK1100_1.TcTerminals210_1BK1250.A_0250_KL_2828_8_Ch_Output_with_Protection_24V_2_0_A_2_wire.Channel_4.Output <-> Channel 4/Output
//     PlcTask Outputs/GVL_iXlinker.EtherCAT_Master_BKCUCX.TcTerminals210_EK1100_1.TcTerminals210_1BK1250.A_0250_KL_2828_8_Ch_Output_with_Protection_24V_2_0_A_2_wire.Channel_5.Output <-> Channel 5/Output
//     PlcTask Outputs/GVL_iXlinker.EtherCAT_Master_BKCUCX.TcTerminals210_EK1100_1.TcTerminals210_1BK1250.A_0250_KL_2828_8_Ch_Output_with_Protection_24V_2_0_A_2_wire.Channel_6.Output <-> Channel 6/Output
//     PlcTask Outputs/GVL_iXlinker.EtherCAT_Master_BKCUCX.TcTerminals210_EK1100_1.TcTerminals210_1BK1250.A_0250_KL_2828_8_Ch_Output_with_Protection_24V_2_0_A_2_wire.Channel_7.Output <-> Channel 7/Output
//     PlcTask Outputs/GVL_iXlinker.EtherCAT_Master_BKCUCX.TcTerminals210_EK1100_1.TcTerminals210_1BK1250.A_0250_KL_2828_8_Ch_Output_with_Protection_24V_2_0_A_2_wire.Channel_8.Output <-> Channel 8/Output
//   PLC/PLC Instance <-> EtherCAT Master BKCUCX/TcTerminals210_EK1100_1/TcTerminals210_1BK1250/A_0251(KL 2809, 16 Ch. Output (24V, 0.5 A))
//     PlcTask Outputs/GVL_iXlinker.EtherCAT_Master_BKCUCX.TcTerminals210_EK1100_1.TcTerminals210_1BK1250.A_0251_KL_2809_16_Ch_Output_24V_0_5_A.Channel_1.Output <-> Channel 1/Output
//     PlcTask Outputs/GVL_iXlinker.EtherCAT_Master_BKCUCX.TcTerminals210_EK1100_1.TcTerminals210_1BK1250.A_0251_KL_2809_16_Ch_Output_24V_0_5_A.Channel_2.Output <-> Channel 2/Output
//     PlcTask Outputs/GVL_iXlinker.EtherCAT_Master_BKCUCX.TcTerminals210_EK1100_1.TcTerminals210_1BK1250.A_0251_KL_2809_16_Ch_Output_24V_0_5_A.Channel_3.Output <-> Channel 3/Output
//     PlcTask Outputs/GVL_iXlinker.EtherCAT_Master_BKCUCX.TcTerminals210_EK1100_1.TcTerminals210_1BK1250.A_0251_KL_2809_16_Ch_Output_24V_0_5_A.Channel_4.Output <-> Channel 4/Output
//     PlcTask Outputs/GVL_iXlinker.EtherCAT_Master_BKCUCX.TcTerminals210_EK1100_1.TcTerminals210_1BK1250.A_0251_KL_2809_16_Ch_Output_24V_0_5_A.Channel_5.Output <-> Channel 5/Output
//     PlcTask Outputs/GVL_iXlinker.EtherCAT_Master_BKCUCX.TcTerminals210_EK1100_1.TcTerminals210_1BK1250.A_0251_KL_2809_16_Ch_Output_24V_0_5_A.Channel_6.Output <-> Channel 6/Output
//     PlcTask Outputs/GVL_iXlinker.EtherCAT_Master_BKCUCX.TcTerminals210_EK1100_1.TcTerminals210_1BK1250.A_0251_KL_2809_16_Ch_Output_24V_0_5_A.Channel_7.Output <-> Channel 7/Output
//     PlcTask Outputs/GVL_iXlinker.EtherCAT_Master_BKCUCX.TcTerminals210_EK1100_1.TcTerminals210_1BK1250.A_0251_KL_2809_16_Ch_Output_24V_0_5_A.Channel_8.Output <-> Channel 8/Output
//     PlcTask Outputs/GVL_iXlinker.EtherCAT_Master_BKCUCX.TcTerminals210_EK1100_1.TcTerminals210_1BK1250.A_0251_KL_2809_16_Ch_Output_24V_0_5_A.Channel_9.Output <-> Channel 9/Output
//     PlcTask Outputs/GVL_iXlinker.EtherCAT_Master_BKCUCX.TcTerminals210_EK1100_1.TcTerminals210_1BK1250.A_0251_KL_2809_16_Ch_Output_24V_0_5_A.Channel_10.Output <-> Channel 10/Output
//     PlcTask Outputs/GVL_iXlinker.EtherCAT_Master_BKCUCX.TcTerminals210_EK1100_1.TcTerminals210_1BK1250.A_0251_KL_2809_16_Ch_Output_24V_0_5_A.Channel_11.Output <-> Channel 11/Output
//     PlcTask Outputs/GVL_iXlinker.EtherCAT_Master_BKCUCX.TcTerminals210_EK1100_1.TcTerminals210_1BK1250.A_0251_KL_2809_16_Ch_Output_24V_0_5_A.Channel_12.Output <-> Channel 12/Output
//     PlcTask Outputs/GVL_iXlinker.EtherCAT_Master_BKCUCX.TcTerminals210_EK1100_1.TcTerminals210_1BK1250.A_0251_KL_2809_16_Ch_Output_24V_0_5_A.Channel_13.Output <-> Channel 13/Output
//     PlcTask Outputs/GVL_iXlinker.EtherCAT_Master_BKCUCX.TcTerminals210_EK1100_1.TcTerminals210_1BK1250.A_0251_KL_2809_16_Ch_Output_24V_0_5_A.Channel_14.Output <-> Channel 14/Output
//     PlcTask Outputs/GVL_iXlinker.EtherCAT_Master_BKCUCX.TcTerminals210_EK1100_1.TcTerminals210_1BK1250.A_0251_KL_2809_16_Ch_Output_24V_0_5_A.Channel_15.Output <-> Channel 15/Output
//     PlcTask Outputs/GVL_iXlinker.EtherCAT_Master_BKCUCX.TcTerminals210_EK1100_1.TcTerminals210_1BK1250.A_0251_KL_2809_16_Ch_Output_24V_0_5_A.Channel_16.Output <-> Channel 16/Output
//   PLC/PLC Instance <-> EtherCAT Master BKCUCX/TcTerminals210_EK1100_1/TcTerminals210_1BK1250/A_0252(KL 2872, 16 Ch. Output (flat-ribbon cable, 24V, 0.5 A))
//     PlcTask Outputs/GVL_iXlinker.EtherCAT_Master_BKCUCX.TcTerminals210_EK1100_1.TcTerminals210_1BK1250.A_0252_KL_2872_16_Ch_Output_flat_ribbon_cable_24V_0_5_A.Channel_1.Output <-> Channel 1/Output
//     PlcTask Outputs/GVL_iXlinker.EtherCAT_Master_BKCUCX.TcTerminals210_EK1100_1.TcTerminals210_1BK1250.A_0252_KL_2872_16_Ch_Output_flat_ribbon_cable_24V_0_5_A.Channel_2.Output <-> Channel 2/Output
//     PlcTask Outputs/GVL_iXlinker.EtherCAT_Master_BKCUCX.TcTerminals210_EK1100_1.TcTerminals210_1BK1250.A_0252_KL_2872_16_Ch_Output_flat_ribbon_cable_24V_0_5_A.Channel_3.Output <-> Channel 3/Output
//     PlcTask Outputs/GVL_iXlinker.EtherCAT_Master_BKCUCX.TcTerminals210_EK1100_1.TcTerminals210_1BK1250.A_0252_KL_2872_16_Ch_Output_flat_ribbon_cable_24V_0_5_A.Channel_4.Output <-> Channel 4/Output
//     PlcTask Outputs/GVL_iXlinker.EtherCAT_Master_BKCUCX.TcTerminals210_EK1100_1.TcTerminals210_1BK1250.A_0252_KL_2872_16_Ch_Output_flat_ribbon_cable_24V_0_5_A.Channel_5.Output <-> Channel 5/Output
//     PlcTask Outputs/GVL_iXlinker.EtherCAT_Master_BKCUCX.TcTerminals210_EK1100_1.TcTerminals210_1BK1250.A_0252_KL_2872_16_Ch_Output_flat_ribbon_cable_24V_0_5_A.Channel_6.Output <-> Channel 6/Output
//     PlcTask Outputs/GVL_iXlinker.EtherCAT_Master_BKCUCX.TcTerminals210_EK1100_1.TcTerminals210_1BK1250.A_0252_KL_2872_16_Ch_Output_flat_ribbon_cable_24V_0_5_A.Channel_7.Output <-> Channel 7/Output
//     PlcTask Outputs/GVL_iXlinker.EtherCAT_Master_BKCUCX.TcTerminals210_EK1100_1.TcTerminals210_1BK1250.A_0252_KL_2872_16_Ch_Output_flat_ribbon_cable_24V_0_5_A.Channel_8.Output <-> Channel 8/Output
//     PlcTask Outputs/GVL_iXlinker.EtherCAT_Master_BKCUCX.TcTerminals210_EK1100_1.TcTerminals210_1BK1250.A_0252_KL_2872_16_Ch_Output_flat_ribbon_cable_24V_0_5_A.Channel_9.Output <-> Channel 9/Output
//     PlcTask Outputs/GVL_iXlinker.EtherCAT_Master_BKCUCX.TcTerminals210_EK1100_1.TcTerminals210_1BK1250.A_0252_KL_2872_16_Ch_Output_flat_ribbon_cable_24V_0_5_A.Channel_10.Output <-> Channel 10/Output
//     PlcTask Outputs/GVL_iXlinker.EtherCAT_Master_BKCUCX.TcTerminals210_EK1100_1.TcTerminals210_1BK1250.A_0252_KL_2872_16_Ch_Output_flat_ribbon_cable_24V_0_5_A.Channel_11.Output <-> Channel 11/Output
//     PlcTask Outputs/GVL_iXlinker.EtherCAT_Master_BKCUCX.TcTerminals210_EK1100_1.TcTerminals210_1BK1250.A_0252_KL_2872_16_Ch_Output_flat_ribbon_cable_24V_0_5_A.Channel_12.Output <-> Channel 12/Output
//     PlcTask Outputs/GVL_iXlinker.EtherCAT_Master_BKCUCX.TcTerminals210_EK1100_1.TcTerminals210_1BK1250.A_0252_KL_2872_16_Ch_Output_flat_ribbon_cable_24V_0_5_A.Channel_13.Output <-> Channel 13/Output
//     PlcTask Outputs/GVL_iXlinker.EtherCAT_Master_BKCUCX.TcTerminals210_EK1100_1.TcTerminals210_1BK1250.A_0252_KL_2872_16_Ch_Output_flat_ribbon_cable_24V_0_5_A.Channel_14.Output <-> Channel 14/Output
//     PlcTask Outputs/GVL_iXlinker.EtherCAT_Master_BKCUCX.TcTerminals210_EK1100_1.TcTerminals210_1BK1250.A_0252_KL_2872_16_Ch_Output_flat_ribbon_cable_24V_0_5_A.Channel_15.Output <-> Channel 15/Output
//     PlcTask Outputs/GVL_iXlinker.EtherCAT_Master_BKCUCX.TcTerminals210_EK1100_1.TcTerminals210_1BK1250.A_0252_KL_2872_16_Ch_Output_flat_ribbon_cable_24V_0_5_A.Channel_16.Output <-> Channel 16/Output
//   PLC/PLC Instance <-> EtherCAT Master BKCUCX/TcTerminals210_EK1100_1/TcTerminals210_1BK1250/A_0253(KL 2889, 16 Ch. Output (24V ground switching, 0.5 A))
//     PlcTask Outputs/GVL_iXlinker.EtherCAT_Master_BKCUCX.TcTerminals210_EK1100_1.TcTerminals210_1BK1250.A_0253_KL_2889_16_Ch_Output_24V_ground_switching_0_5_A.Channel_1.Output <-> Channel 1/Output
//     PlcTask Outputs/GVL_iXlinker.EtherCAT_Master_BKCUCX.TcTerminals210_EK1100_1.TcTerminals210_1BK1250.A_0253_KL_2889_16_Ch_Output_24V_ground_switching_0_5_A.Channel_2.Output <-> Channel 2/Output
//     PlcTask Outputs/GVL_iXlinker.EtherCAT_Master_BKCUCX.TcTerminals210_EK1100_1.TcTerminals210_1BK1250.A_0253_KL_2889_16_Ch_Output_24V_ground_switching_0_5_A.Channel_3.Output <-> Channel 3/Output
//     PlcTask Outputs/GVL_iXlinker.EtherCAT_Master_BKCUCX.TcTerminals210_EK1100_1.TcTerminals210_1BK1250.A_0253_KL_2889_16_Ch_Output_24V_ground_switching_0_5_A.Channel_4.Output <-> Channel 4/Output
//     PlcTask Outputs/GVL_iXlinker.EtherCAT_Master_BKCUCX.TcTerminals210_EK1100_1.TcTerminals210_1BK1250.A_0253_KL_2889_16_Ch_Output_24V_ground_switching_0_5_A.Channel_5.Output <-> Channel 5/Output
//     PlcTask Outputs/GVL_iXlinker.EtherCAT_Master_BKCUCX.TcTerminals210_EK1100_1.TcTerminals210_1BK1250.A_0253_KL_2889_16_Ch_Output_24V_ground_switching_0_5_A.Channel_6.Output <-> Channel 6/Output
//     PlcTask Outputs/GVL_iXlinker.EtherCAT_Master_BKCUCX.TcTerminals210_EK1100_1.TcTerminals210_1BK1250.A_0253_KL_2889_16_Ch_Output_24V_ground_switching_0_5_A.Channel_7.Output <-> Channel 7/Output
//     PlcTask Outputs/GVL_iXlinker.EtherCAT_Master_BKCUCX.TcTerminals210_EK1100_1.TcTerminals210_1BK1250.A_0253_KL_2889_16_Ch_Output_24V_ground_switching_0_5_A.Channel_8.Output <-> Channel 8/Output
//     PlcTask Outputs/GVL_iXlinker.EtherCAT_Master_BKCUCX.TcTerminals210_EK1100_1.TcTerminals210_1BK1250.A_0253_KL_2889_16_Ch_Output_24V_ground_switching_0_5_A.Channel_9.Output <-> Channel 9/Output
//     PlcTask Outputs/GVL_iXlinker.EtherCAT_Master_BKCUCX.TcTerminals210_EK1100_1.TcTerminals210_1BK1250.A_0253_KL_2889_16_Ch_Output_24V_ground_switching_0_5_A.Channel_10.Output <-> Channel 10/Output
//     PlcTask Outputs/GVL_iXlinker.EtherCAT_Master_BKCUCX.TcTerminals210_EK1100_1.TcTerminals210_1BK1250.A_0253_KL_2889_16_Ch_Output_24V_ground_switching_0_5_A.Channel_11.Output <-> Channel 11/Output
//     PlcTask Outputs/GVL_iXlinker.EtherCAT_Master_BKCUCX.TcTerminals210_EK1100_1.TcTerminals210_1BK1250.A_0253_KL_2889_16_Ch_Output_24V_ground_switching_0_5_A.Channel_12.Output <-> Channel 12/Output
//     PlcTask Outputs/GVL_iXlinker.EtherCAT_Master_BKCUCX.TcTerminals210_EK1100_1.TcTerminals210_1BK1250.A_0253_KL_2889_16_Ch_Output_24V_ground_switching_0_5_A.Channel_13.Output <-> Channel 13/Output
//     PlcTask Outputs/GVL_iXlinker.EtherCAT_Master_BKCUCX.TcTerminals210_EK1100_1.TcTerminals210_1BK1250.A_0253_KL_2889_16_Ch_Output_24V_ground_switching_0_5_A.Channel_14.Output <-> Channel 14/Output
//     PlcTask Outputs/GVL_iXlinker.EtherCAT_Master_BKCUCX.TcTerminals210_EK1100_1.TcTerminals210_1BK1250.A_0253_KL_2889_16_Ch_Output_24V_ground_switching_0_5_A.Channel_15.Output <-> Channel 15/Output
//     PlcTask Outputs/GVL_iXlinker.EtherCAT_Master_BKCUCX.TcTerminals210_EK1100_1.TcTerminals210_1BK1250.A_0253_KL_2889_16_Ch_Output_24V_ground_switching_0_5_A.Channel_16.Output <-> Channel 16/Output
//   PLC/PLC Instance <-> EtherCAT Master BKCUCX/TcTerminals210_EK1100_1/TcTerminals210_1BK1250/A_0254(KL 2904, 4 Ch. Safety Output)
//     PlcTask Inputs/GVL_iXlinker.EtherCAT_Master_BKCUCX.TcTerminals210_EK1100_1.TcTerminals210_1BK1250.A_0254_KL_2904_4_Ch_Safety_Output.Channel_1.Safety_In <-> Channel 1/Safety In
//     PlcTask Outputs/GVL_iXlinker.EtherCAT_Master_BKCUCX.TcTerminals210_EK1100_1.TcTerminals210_1BK1250.A_0254_KL_2904_4_Ch_Safety_Output.Channel_1.Safety_Out <-> Channel 1/Safety Out
//   PLC/PLC Instance <-> EtherCAT Master BKCUCX/TcTerminals210_EK1100_1/TcTerminals210_1BK1250/A_0255(KM 2002, 16 Ch. Output (24V, 0.5 A))
//     PlcTask Outputs/GVL_iXlinker.EtherCAT_Master_BKCUCX.TcTerminals210_EK1100_1.TcTerminals210_1BK1250.A_0255_KM_2002_16_Ch_Output_24V_0_5_A.Channel_1.Output <-> Channel 1/Output
//     PlcTask Outputs/GVL_iXlinker.EtherCAT_Master_BKCUCX.TcTerminals210_EK1100_1.TcTerminals210_1BK1250.A_0255_KM_2002_16_Ch_Output_24V_0_5_A.Channel_2.Output <-> Channel 2/Output
//     PlcTask Outputs/GVL_iXlinker.EtherCAT_Master_BKCUCX.TcTerminals210_EK1100_1.TcTerminals210_1BK1250.A_0255_KM_2002_16_Ch_Output_24V_0_5_A.Channel_3.Output <-> Channel 3/Output
//     PlcTask Outputs/GVL_iXlinker.EtherCAT_Master_BKCUCX.TcTerminals210_EK1100_1.TcTerminals210_1BK1250.A_0255_KM_2002_16_Ch_Output_24V_0_5_A.Channel_4.Output <-> Channel 4/Output
//     PlcTask Outputs/GVL_iXlinker.EtherCAT_Master_BKCUCX.TcTerminals210_EK1100_1.TcTerminals210_1BK1250.A_0255_KM_2002_16_Ch_Output_24V_0_5_A.Channel_5.Output <-> Channel 5/Output
//     PlcTask Outputs/GVL_iXlinker.EtherCAT_Master_BKCUCX.TcTerminals210_EK1100_1.TcTerminals210_1BK1250.A_0255_KM_2002_16_Ch_Output_24V_0_5_A.Channel_6.Output <-> Channel 6/Output
//     PlcTask Outputs/GVL_iXlinker.EtherCAT_Master_BKCUCX.TcTerminals210_EK1100_1.TcTerminals210_1BK1250.A_0255_KM_2002_16_Ch_Output_24V_0_5_A.Channel_7.Output <-> Channel 7/Output
//     PlcTask Outputs/GVL_iXlinker.EtherCAT_Master_BKCUCX.TcTerminals210_EK1100_1.TcTerminals210_1BK1250.A_0255_KM_2002_16_Ch_Output_24V_0_5_A.Channel_8.Output <-> Channel 8/Output
//     PlcTask Outputs/GVL_iXlinker.EtherCAT_Master_BKCUCX.TcTerminals210_EK1100_1.TcTerminals210_1BK1250.A_0255_KM_2002_16_Ch_Output_24V_0_5_A.Channel_9.Output <-> Channel 9/Output
//     PlcTask Outputs/GVL_iXlinker.EtherCAT_Master_BKCUCX.TcTerminals210_EK1100_1.TcTerminals210_1BK1250.A_0255_KM_2002_16_Ch_Output_24V_0_5_A.Channel_10.Output <-> Channel 10/Output
//     PlcTask Outputs/GVL_iXlinker.EtherCAT_Master_BKCUCX.TcTerminals210_EK1100_1.TcTerminals210_1BK1250.A_0255_KM_2002_16_Ch_Output_24V_0_5_A.Channel_11.Output <-> Channel 11/Output
//     PlcTask Outputs/GVL_iXlinker.EtherCAT_Master_BKCUCX.TcTerminals210_EK1100_1.TcTerminals210_1BK1250.A_0255_KM_2002_16_Ch_Output_24V_0_5_A.Channel_12.Output <-> Channel 12/Output
//     PlcTask Outputs/GVL_iXlinker.EtherCAT_Master_BKCUCX.TcTerminals210_EK1100_1.TcTerminals210_1BK1250.A_0255_KM_2002_16_Ch_Output_24V_0_5_A.Channel_13.Output <-> Channel 13/Output
//     PlcTask Outputs/GVL_iXlinker.EtherCAT_Master_BKCUCX.TcTerminals210_EK1100_1.TcTerminals210_1BK1250.A_0255_KM_2002_16_Ch_Output_24V_0_5_A.Channel_14.Output <-> Channel 14/Output
//     PlcTask Outputs/GVL_iXlinker.EtherCAT_Master_BKCUCX.TcTerminals210_EK1100_1.TcTerminals210_1BK1250.A_0255_KM_2002_16_Ch_Output_24V_0_5_A.Channel_15.Output <-> Channel 15/Output
//     PlcTask Outputs/GVL_iXlinker.EtherCAT_Master_BKCUCX.TcTerminals210_EK1100_1.TcTerminals210_1BK1250.A_0255_KM_2002_16_Ch_Output_24V_0_5_A.Channel_16.Output <-> Channel 16/Output
//   PLC/PLC Instance <-> EtherCAT Master BKCUCX/TcTerminals210_EK1100_1/TcTerminals210_1BK1250/A_0256(KM 2004, 32 Ch. Output (24V, 0.5 A))
//     PlcTask Outputs/GVL_iXlinker.EtherCAT_Master_BKCUCX.TcTerminals210_EK1100_1.TcTerminals210_1BK1250.A_0256_KM_2004_32_Ch_Output_24V_0_5_A.Channel_1.Output <-> Channel 1/Output
//     PlcTask Outputs/GVL_iXlinker.EtherCAT_Master_BKCUCX.TcTerminals210_EK1100_1.TcTerminals210_1BK1250.A_0256_KM_2004_32_Ch_Output_24V_0_5_A.Channel_2.Output <-> Channel 2/Output
//     PlcTask Outputs/GVL_iXlinker.EtherCAT_Master_BKCUCX.TcTerminals210_EK1100_1.TcTerminals210_1BK1250.A_0256_KM_2004_32_Ch_Output_24V_0_5_A.Channel_3.Output <-> Channel 3/Output
//     PlcTask Outputs/GVL_iXlinker.EtherCAT_Master_BKCUCX.TcTerminals210_EK1100_1.TcTerminals210_1BK1250.A_0256_KM_2004_32_Ch_Output_24V_0_5_A.Channel_4.Output <-> Channel 4/Output
//     PlcTask Outputs/GVL_iXlinker.EtherCAT_Master_BKCUCX.TcTerminals210_EK1100_1.TcTerminals210_1BK1250.A_0256_KM_2004_32_Ch_Output_24V_0_5_A.Channel_5.Output <-> Channel 5/Output
//     PlcTask Outputs/GVL_iXlinker.EtherCAT_Master_BKCUCX.TcTerminals210_EK1100_1.TcTerminals210_1BK1250.A_0256_KM_2004_32_Ch_Output_24V_0_5_A.Channel_6.Output <-> Channel 6/Output
//     PlcTask Outputs/GVL_iXlinker.EtherCAT_Master_BKCUCX.TcTerminals210_EK1100_1.TcTerminals210_1BK1250.A_0256_KM_2004_32_Ch_Output_24V_0_5_A.Channel_7.Output <-> Channel 7/Output
//     PlcTask Outputs/GVL_iXlinker.EtherCAT_Master_BKCUCX.TcTerminals210_EK1100_1.TcTerminals210_1BK1250.A_0256_KM_2004_32_Ch_Output_24V_0_5_A.Channel_8.Output <-> Channel 8/Output
//     PlcTask Outputs/GVL_iXlinker.EtherCAT_Master_BKCUCX.TcTerminals210_EK1100_1.TcTerminals210_1BK1250.A_0256_KM_2004_32_Ch_Output_24V_0_5_A.Channel_9.Output <-> Channel 9/Output
//     PlcTask Outputs/GVL_iXlinker.EtherCAT_Master_BKCUCX.TcTerminals210_EK1100_1.TcTerminals210_1BK1250.A_0256_KM_2004_32_Ch_Output_24V_0_5_A.Channel_10.Output <-> Channel 10/Output
//     PlcTask Outputs/GVL_iXlinker.EtherCAT_Master_BKCUCX.TcTerminals210_EK1100_1.TcTerminals210_1BK1250.A_0256_KM_2004_32_Ch_Output_24V_0_5_A.Channel_11.Output <-> Channel 11/Output
//     PlcTask Outputs/GVL_iXlinker.EtherCAT_Master_BKCUCX.TcTerminals210_EK1100_1.TcTerminals210_1BK1250.A_0256_KM_2004_32_Ch_Output_24V_0_5_A.Channel_12.Output <-> Channel 12/Output
//     PlcTask Outputs/GVL_iXlinker.EtherCAT_Master_BKCUCX.TcTerminals210_EK1100_1.TcTerminals210_1BK1250.A_0256_KM_2004_32_Ch_Output_24V_0_5_A.Channel_13.Output <-> Channel 13/Output
//     PlcTask Outputs/GVL_iXlinker.EtherCAT_Master_BKCUCX.TcTerminals210_EK1100_1.TcTerminals210_1BK1250.A_0256_KM_2004_32_Ch_Output_24V_0_5_A.Channel_14.Output <-> Channel 14/Output
//     PlcTask Outputs/GVL_iXlinker.EtherCAT_Master_BKCUCX.TcTerminals210_EK1100_1.TcTerminals210_1BK1250.A_0256_KM_2004_32_Ch_Output_24V_0_5_A.Channel_15.Output <-> Channel 15/Output
//     PlcTask Outputs/GVL_iXlinker.EtherCAT_Master_BKCUCX.TcTerminals210_EK1100_1.TcTerminals210_1BK1250.A_0256_KM_2004_32_Ch_Output_24V_0_5_A.Channel_16.Output <-> Channel 16/Output
//     PlcTask Outputs/GVL_iXlinker.EtherCAT_Master_BKCUCX.TcTerminals210_EK1100_1.TcTerminals210_1BK1250.A_0256_KM_2004_32_Ch_Output_24V_0_5_A.Channel_17.Output <-> Channel 17/Output
//     PlcTask Outputs/GVL_iXlinker.EtherCAT_Master_BKCUCX.TcTerminals210_EK1100_1.TcTerminals210_1BK1250.A_0256_KM_2004_32_Ch_Output_24V_0_5_A.Channel_18.Output <-> Channel 18/Output
//     PlcTask Outputs/GVL_iXlinker.EtherCAT_Master_BKCUCX.TcTerminals210_EK1100_1.TcTerminals210_1BK1250.A_0256_KM_2004_32_Ch_Output_24V_0_5_A.Channel_19.Output <-> Channel 19/Output
//     PlcTask Outputs/GVL_iXlinker.EtherCAT_Master_BKCUCX.TcTerminals210_EK1100_1.TcTerminals210_1BK1250.A_0256_KM_2004_32_Ch_Output_24V_0_5_A.Channel_20.Output <-> Channel 20/Output
//     PlcTask Outputs/GVL_iXlinker.EtherCAT_Master_BKCUCX.TcTerminals210_EK1100_1.TcTerminals210_1BK1250.A_0256_KM_2004_32_Ch_Output_24V_0_5_A.Channel_21.Output <-> Channel 21/Output
//     PlcTask Outputs/GVL_iXlinker.EtherCAT_Master_BKCUCX.TcTerminals210_EK1100_1.TcTerminals210_1BK1250.A_0256_KM_2004_32_Ch_Output_24V_0_5_A.Channel_22.Output <-> Channel 22/Output
//     PlcTask Outputs/GVL_iXlinker.EtherCAT_Master_BKCUCX.TcTerminals210_EK1100_1.TcTerminals210_1BK1250.A_0256_KM_2004_32_Ch_Output_24V_0_5_A.Channel_23.Output <-> Channel 23/Output
//     PlcTask Outputs/GVL_iXlinker.EtherCAT_Master_BKCUCX.TcTerminals210_EK1100_1.TcTerminals210_1BK1250.A_0256_KM_2004_32_Ch_Output_24V_0_5_A.Channel_24.Output <-> Channel 24/Output
//     PlcTask Outputs/GVL_iXlinker.EtherCAT_Master_BKCUCX.TcTerminals210_EK1100_1.TcTerminals210_1BK1250.A_0256_KM_2004_32_Ch_Output_24V_0_5_A.Channel_25.Output <-> Channel 25/Output
//     PlcTask Outputs/GVL_iXlinker.EtherCAT_Master_BKCUCX.TcTerminals210_EK1100_1.TcTerminals210_1BK1250.A_0256_KM_2004_32_Ch_Output_24V_0_5_A.Channel_26.Output <-> Channel 26/Output
//     PlcTask Outputs/GVL_iXlinker.EtherCAT_Master_BKCUCX.TcTerminals210_EK1100_1.TcTerminals210_1BK1250.A_0256_KM_2004_32_Ch_Output_24V_0_5_A.Channel_27.Output <-> Channel 27/Output
//     PlcTask Outputs/GVL_iXlinker.EtherCAT_Master_BKCUCX.TcTerminals210_EK1100_1.TcTerminals210_1BK1250.A_0256_KM_2004_32_Ch_Output_24V_0_5_A.Channel_28.Output <-> Channel 28/Output
//     PlcTask Outputs/GVL_iXlinker.EtherCAT_Master_BKCUCX.TcTerminals210_EK1100_1.TcTerminals210_1BK1250.A_0256_KM_2004_32_Ch_Output_24V_0_5_A.Channel_29.Output <-> Channel 29/Output
//     PlcTask Outputs/GVL_iXlinker.EtherCAT_Master_BKCUCX.TcTerminals210_EK1100_1.TcTerminals210_1BK1250.A_0256_KM_2004_32_Ch_Output_24V_0_5_A.Channel_30.Output <-> Channel 30/Output
//     PlcTask Outputs/GVL_iXlinker.EtherCAT_Master_BKCUCX.TcTerminals210_EK1100_1.TcTerminals210_1BK1250.A_0256_KM_2004_32_Ch_Output_24V_0_5_A.Channel_31.Output <-> Channel 31/Output
//     PlcTask Outputs/GVL_iXlinker.EtherCAT_Master_BKCUCX.TcTerminals210_EK1100_1.TcTerminals210_1BK1250.A_0256_KM_2004_32_Ch_Output_24V_0_5_A.Channel_32.Output <-> Channel 32/Output
//   PLC/PLC Instance <-> EtherCAT Master BKCUCX/TcTerminals210_EK1100_1/TcTerminals210_1BK1250/A_0257(KM 2008, 64 Ch. Output (24V, 0.5 A))
//     PlcTask Outputs/GVL_iXlinker.EtherCAT_Master_BKCUCX.TcTerminals210_EK1100_1.TcTerminals210_1BK1250.A_0257_KM_2008_64_Ch_Output_24V_0_5_A.Channel_1.Output <-> Channel 1/Output
//     PlcTask Outputs/GVL_iXlinker.EtherCAT_Master_BKCUCX.TcTerminals210_EK1100_1.TcTerminals210_1BK1250.A_0257_KM_2008_64_Ch_Output_24V_0_5_A.Channel_2.Output <-> Channel 2/Output
//     PlcTask Outputs/GVL_iXlinker.EtherCAT_Master_BKCUCX.TcTerminals210_EK1100_1.TcTerminals210_1BK1250.A_0257_KM_2008_64_Ch_Output_24V_0_5_A.Channel_3.Output <-> Channel 3/Output
//     PlcTask Outputs/GVL_iXlinker.EtherCAT_Master_BKCUCX.TcTerminals210_EK1100_1.TcTerminals210_1BK1250.A_0257_KM_2008_64_Ch_Output_24V_0_5_A.Channel_4.Output <-> Channel 4/Output
//     PlcTask Outputs/GVL_iXlinker.EtherCAT_Master_BKCUCX.TcTerminals210_EK1100_1.TcTerminals210_1BK1250.A_0257_KM_2008_64_Ch_Output_24V_0_5_A.Channel_5.Output <-> Channel 5/Output
//     PlcTask Outputs/GVL_iXlinker.EtherCAT_Master_BKCUCX.TcTerminals210_EK1100_1.TcTerminals210_1BK1250.A_0257_KM_2008_64_Ch_Output_24V_0_5_A.Channel_6.Output <-> Channel 6/Output
//     PlcTask Outputs/GVL_iXlinker.EtherCAT_Master_BKCUCX.TcTerminals210_EK1100_1.TcTerminals210_1BK1250.A_0257_KM_2008_64_Ch_Output_24V_0_5_A.Channel_7.Output <-> Channel 7/Output
//     PlcTask Outputs/GVL_iXlinker.EtherCAT_Master_BKCUCX.TcTerminals210_EK1100_1.TcTerminals210_1BK1250.A_0257_KM_2008_64_Ch_Output_24V_0_5_A.Channel_8.Output <-> Channel 8/Output
//     PlcTask Outputs/GVL_iXlinker.EtherCAT_Master_BKCUCX.TcTerminals210_EK1100_1.TcTerminals210_1BK1250.A_0257_KM_2008_64_Ch_Output_24V_0_5_A.Channel_9.Output <-> Channel 9/Output
//     PlcTask Outputs/GVL_iXlinker.EtherCAT_Master_BKCUCX.TcTerminals210_EK1100_1.TcTerminals210_1BK1250.A_0257_KM_2008_64_Ch_Output_24V_0_5_A.Channel_10.Output <-> Channel 10/Output
//     PlcTask Outputs/GVL_iXlinker.EtherCAT_Master_BKCUCX.TcTerminals210_EK1100_1.TcTerminals210_1BK1250.A_0257_KM_2008_64_Ch_Output_24V_0_5_A.Channel_11.Output <-> Channel 11/Output
//     PlcTask Outputs/GVL_iXlinker.EtherCAT_Master_BKCUCX.TcTerminals210_EK1100_1.TcTerminals210_1BK1250.A_0257_KM_2008_64_Ch_Output_24V_0_5_A.Channel_12.Output <-> Channel 12/Output
//     PlcTask Outputs/GVL_iXlinker.EtherCAT_Master_BKCUCX.TcTerminals210_EK1100_1.TcTerminals210_1BK1250.A_0257_KM_2008_64_Ch_Output_24V_0_5_A.Channel_13.Output <-> Channel 13/Output
//     PlcTask Outputs/GVL_iXlinker.EtherCAT_Master_BKCUCX.TcTerminals210_EK1100_1.TcTerminals210_1BK1250.A_0257_KM_2008_64_Ch_Output_24V_0_5_A.Channel_14.Output <-> Channel 14/Output
//     PlcTask Outputs/GVL_iXlinker.EtherCAT_Master_BKCUCX.TcTerminals210_EK1100_1.TcTerminals210_1BK1250.A_0257_KM_2008_64_Ch_Output_24V_0_5_A.Channel_15.Output <-> Channel 15/Output
//     PlcTask Outputs/GVL_iXlinker.EtherCAT_Master_BKCUCX.TcTerminals210_EK1100_1.TcTerminals210_1BK1250.A_0257_KM_2008_64_Ch_Output_24V_0_5_A.Channel_16.Output <-> Channel 16/Output
//     PlcTask Outputs/GVL_iXlinker.EtherCAT_Master_BKCUCX.TcTerminals210_EK1100_1.TcTerminals210_1BK1250.A_0257_KM_2008_64_Ch_Output_24V_0_5_A.Channel_17.Output <-> Channel 17/Output
//     PlcTask Outputs/GVL_iXlinker.EtherCAT_Master_BKCUCX.TcTerminals210_EK1100_1.TcTerminals210_1BK1250.A_0257_KM_2008_64_Ch_Output_24V_0_5_A.Channel_18.Output <-> Channel 18/Output
//     PlcTask Outputs/GVL_iXlinker.EtherCAT_Master_BKCUCX.TcTerminals210_EK1100_1.TcTerminals210_1BK1250.A_0257_KM_2008_64_Ch_Output_24V_0_5_A.Channel_19.Output <-> Channel 19/Output
//     PlcTask Outputs/GVL_iXlinker.EtherCAT_Master_BKCUCX.TcTerminals210_EK1100_1.TcTerminals210_1BK1250.A_0257_KM_2008_64_Ch_Output_24V_0_5_A.Channel_20.Output <-> Channel 20/Output
//     PlcTask Outputs/GVL_iXlinker.EtherCAT_Master_BKCUCX.TcTerminals210_EK1100_1.TcTerminals210_1BK1250.A_0257_KM_2008_64_Ch_Output_24V_0_5_A.Channel_21.Output <-> Channel 21/Output
//     PlcTask Outputs/GVL_iXlinker.EtherCAT_Master_BKCUCX.TcTerminals210_EK1100_1.TcTerminals210_1BK1250.A_0257_KM_2008_64_Ch_Output_24V_0_5_A.Channel_22.Output <-> Channel 22/Output
//     PlcTask Outputs/GVL_iXlinker.EtherCAT_Master_BKCUCX.TcTerminals210_EK1100_1.TcTerminals210_1BK1250.A_0257_KM_2008_64_Ch_Output_24V_0_5_A.Channel_23.Output <-> Channel 23/Output
//     PlcTask Outputs/GVL_iXlinker.EtherCAT_Master_BKCUCX.TcTerminals210_EK1100_1.TcTerminals210_1BK1250.A_0257_KM_2008_64_Ch_Output_24V_0_5_A.Channel_24.Output <-> Channel 24/Output
//     PlcTask Outputs/GVL_iXlinker.EtherCAT_Master_BKCUCX.TcTerminals210_EK1100_1.TcTerminals210_1BK1250.A_0257_KM_2008_64_Ch_Output_24V_0_5_A.Channel_25.Output <-> Channel 25/Output
//     PlcTask Outputs/GVL_iXlinker.EtherCAT_Master_BKCUCX.TcTerminals210_EK1100_1.TcTerminals210_1BK1250.A_0257_KM_2008_64_Ch_Output_24V_0_5_A.Channel_26.Output <-> Channel 26/Output
//     PlcTask Outputs/GVL_iXlinker.EtherCAT_Master_BKCUCX.TcTerminals210_EK1100_1.TcTerminals210_1BK1250.A_0257_KM_2008_64_Ch_Output_24V_0_5_A.Channel_27.Output <-> Channel 27/Output
//     PlcTask Outputs/GVL_iXlinker.EtherCAT_Master_BKCUCX.TcTerminals210_EK1100_1.TcTerminals210_1BK1250.A_0257_KM_2008_64_Ch_Output_24V_0_5_A.Channel_28.Output <-> Channel 28/Output
//     PlcTask Outputs/GVL_iXlinker.EtherCAT_Master_BKCUCX.TcTerminals210_EK1100_1.TcTerminals210_1BK1250.A_0257_KM_2008_64_Ch_Output_24V_0_5_A.Channel_29.Output <-> Channel 29/Output
//     PlcTask Outputs/GVL_iXlinker.EtherCAT_Master_BKCUCX.TcTerminals210_EK1100_1.TcTerminals210_1BK1250.A_0257_KM_2008_64_Ch_Output_24V_0_5_A.Channel_30.Output <-> Channel 30/Output
//     PlcTask Outputs/GVL_iXlinker.EtherCAT_Master_BKCUCX.TcTerminals210_EK1100_1.TcTerminals210_1BK1250.A_0257_KM_2008_64_Ch_Output_24V_0_5_A.Channel_31.Output <-> Channel 31/Output
//     PlcTask Outputs/GVL_iXlinker.EtherCAT_Master_BKCUCX.TcTerminals210_EK1100_1.TcTerminals210_1BK1250.A_0257_KM_2008_64_Ch_Output_24V_0_5_A.Channel_32.Output <-> Channel 32/Output
//     PlcTask Outputs/GVL_iXlinker.EtherCAT_Master_BKCUCX.TcTerminals210_EK1100_1.TcTerminals210_1BK1250.A_0257_KM_2008_64_Ch_Output_24V_0_5_A.Channel_33.Output <-> Channel 33/Output
//     PlcTask Outputs/GVL_iXlinker.EtherCAT_Master_BKCUCX.TcTerminals210_EK1100_1.TcTerminals210_1BK1250.A_0257_KM_2008_64_Ch_Output_24V_0_5_A.Channel_34.Output <-> Channel 34/Output
//     PlcTask Outputs/GVL_iXlinker.EtherCAT_Master_BKCUCX.TcTerminals210_EK1100_1.TcTerminals210_1BK1250.A_0257_KM_2008_64_Ch_Output_24V_0_5_A.Channel_35.Output <-> Channel 35/Output
//     PlcTask Outputs/GVL_iXlinker.EtherCAT_Master_BKCUCX.TcTerminals210_EK1100_1.TcTerminals210_1BK1250.A_0257_KM_2008_64_Ch_Output_24V_0_5_A.Channel_36.Output <-> Channel 36/Output
//     PlcTask Outputs/GVL_iXlinker.EtherCAT_Master_BKCUCX.TcTerminals210_EK1100_1.TcTerminals210_1BK1250.A_0257_KM_2008_64_Ch_Output_24V_0_5_A.Channel_37.Output <-> Channel 37/Output
//     PlcTask Outputs/GVL_iXlinker.EtherCAT_Master_BKCUCX.TcTerminals210_EK1100_1.TcTerminals210_1BK1250.A_0257_KM_2008_64_Ch_Output_24V_0_5_A.Channel_38.Output <-> Channel 38/Output
//     PlcTask Outputs/GVL_iXlinker.EtherCAT_Master_BKCUCX.TcTerminals210_EK1100_1.TcTerminals210_1BK1250.A_0257_KM_2008_64_Ch_Output_24V_0_5_A.Channel_39.Output <-> Channel 39/Output
//     PlcTask Outputs/GVL_iXlinker.EtherCAT_Master_BKCUCX.TcTerminals210_EK1100_1.TcTerminals210_1BK1250.A_0257_KM_2008_64_Ch_Output_24V_0_5_A.Channel_40.Output <-> Channel 40/Output
//     PlcTask Outputs/GVL_iXlinker.EtherCAT_Master_BKCUCX.TcTerminals210_EK1100_1.TcTerminals210_1BK1250.A_0257_KM_2008_64_Ch_Output_24V_0_5_A.Channel_41.Output <-> Channel 41/Output
//     PlcTask Outputs/GVL_iXlinker.EtherCAT_Master_BKCUCX.TcTerminals210_EK1100_1.TcTerminals210_1BK1250.A_0257_KM_2008_64_Ch_Output_24V_0_5_A.Channel_42.Output <-> Channel 42/Output
//     PlcTask Outputs/GVL_iXlinker.EtherCAT_Master_BKCUCX.TcTerminals210_EK1100_1.TcTerminals210_1BK1250.A_0257_KM_2008_64_Ch_Output_24V_0_5_A.Channel_43.Output <-> Channel 43/Output
//     PlcTask Outputs/GVL_iXlinker.EtherCAT_Master_BKCUCX.TcTerminals210_EK1100_1.TcTerminals210_1BK1250.A_0257_KM_2008_64_Ch_Output_24V_0_5_A.Channel_44.Output <-> Channel 44/Output
//     PlcTask Outputs/GVL_iXlinker.EtherCAT_Master_BKCUCX.TcTerminals210_EK1100_1.TcTerminals210_1BK1250.A_0257_KM_2008_64_Ch_Output_24V_0_5_A.Channel_45.Output <-> Channel 45/Output
//     PlcTask Outputs/GVL_iXlinker.EtherCAT_Master_BKCUCX.TcTerminals210_EK1100_1.TcTerminals210_1BK1250.A_0257_KM_2008_64_Ch_Output_24V_0_5_A.Channel_46.Output <-> Channel 46/Output
//     PlcTask Outputs/GVL_iXlinker.EtherCAT_Master_BKCUCX.TcTerminals210_EK1100_1.TcTerminals210_1BK1250.A_0257_KM_2008_64_Ch_Output_24V_0_5_A.Channel_47.Output <-> Channel 47/Output
//     PlcTask Outputs/GVL_iXlinker.EtherCAT_Master_BKCUCX.TcTerminals210_EK1100_1.TcTerminals210_1BK1250.A_0257_KM_2008_64_Ch_Output_24V_0_5_A.Channel_48.Output <-> Channel 48/Output
//     PlcTask Outputs/GVL_iXlinker.EtherCAT_Master_BKCUCX.TcTerminals210_EK1100_1.TcTerminals210_1BK1250.A_0257_KM_2008_64_Ch_Output_24V_0_5_A.Channel_49.Output <-> Channel 49/Output
//     PlcTask Outputs/GVL_iXlinker.EtherCAT_Master_BKCUCX.TcTerminals210_EK1100_1.TcTerminals210_1BK1250.A_0257_KM_2008_64_Ch_Output_24V_0_5_A.Channel_50.Output <-> Channel 50/Output
//     PlcTask Outputs/GVL_iXlinker.EtherCAT_Master_BKCUCX.TcTerminals210_EK1100_1.TcTerminals210_1BK1250.A_0257_KM_2008_64_Ch_Output_24V_0_5_A.Channel_51.Output <-> Channel 51/Output
//     PlcTask Outputs/GVL_iXlinker.EtherCAT_Master_BKCUCX.TcTerminals210_EK1100_1.TcTerminals210_1BK1250.A_0257_KM_2008_64_Ch_Output_24V_0_5_A.Channel_52.Output <-> Channel 52/Output
//     PlcTask Outputs/GVL_iXlinker.EtherCAT_Master_BKCUCX.TcTerminals210_EK1100_1.TcTerminals210_1BK1250.A_0257_KM_2008_64_Ch_Output_24V_0_5_A.Channel_53.Output <-> Channel 53/Output
//     PlcTask Outputs/GVL_iXlinker.EtherCAT_Master_BKCUCX.TcTerminals210_EK1100_1.TcTerminals210_1BK1250.A_0257_KM_2008_64_Ch_Output_24V_0_5_A.Channel_54.Output <-> Channel 54/Output
//     PlcTask Outputs/GVL_iXlinker.EtherCAT_Master_BKCUCX.TcTerminals210_EK1100_1.TcTerminals210_1BK1250.A_0257_KM_2008_64_Ch_Output_24V_0_5_A.Channel_55.Output <-> Channel 55/Output
//     PlcTask Outputs/GVL_iXlinker.EtherCAT_Master_BKCUCX.TcTerminals210_EK1100_1.TcTerminals210_1BK1250.A_0257_KM_2008_64_Ch_Output_24V_0_5_A.Channel_56.Output <-> Channel 56/Output
//     PlcTask Outputs/GVL_iXlinker.EtherCAT_Master_BKCUCX.TcTerminals210_EK1100_1.TcTerminals210_1BK1250.A_0257_KM_2008_64_Ch_Output_24V_0_5_A.Channel_57.Output <-> Channel 57/Output
//     PlcTask Outputs/GVL_iXlinker.EtherCAT_Master_BKCUCX.TcTerminals210_EK1100_1.TcTerminals210_1BK1250.A_0257_KM_2008_64_Ch_Output_24V_0_5_A.Channel_58.Output <-> Channel 58/Output
//     PlcTask Outputs/GVL_iXlinker.EtherCAT_Master_BKCUCX.TcTerminals210_EK1100_1.TcTerminals210_1BK1250.A_0257_KM_2008_64_Ch_Output_24V_0_5_A.Channel_59.Output <-> Channel 59/Output
//     PlcTask Outputs/GVL_iXlinker.EtherCAT_Master_BKCUCX.TcTerminals210_EK1100_1.TcTerminals210_1BK1250.A_0257_KM_2008_64_Ch_Output_24V_0_5_A.Channel_60.Output <-> Channel 60/Output
//     PlcTask Outputs/GVL_iXlinker.EtherCAT_Master_BKCUCX.TcTerminals210_EK1100_1.TcTerminals210_1BK1250.A_0257_KM_2008_64_Ch_Output_24V_0_5_A.Channel_61.Output <-> Channel 61/Output
//     PlcTask Outputs/GVL_iXlinker.EtherCAT_Master_BKCUCX.TcTerminals210_EK1100_1.TcTerminals210_1BK1250.A_0257_KM_2008_64_Ch_Output_24V_0_5_A.Channel_62.Output <-> Channel 62/Output
//     PlcTask Outputs/GVL_iXlinker.EtherCAT_Master_BKCUCX.TcTerminals210_EK1100_1.TcTerminals210_1BK1250.A_0257_KM_2008_64_Ch_Output_24V_0_5_A.Channel_63.Output <-> Channel 63/Output
//     PlcTask Outputs/GVL_iXlinker.EtherCAT_Master_BKCUCX.TcTerminals210_EK1100_1.TcTerminals210_1BK1250.A_0257_KM_2008_64_Ch_Output_24V_0_5_A.Channel_64.Output <-> Channel 64/Output
//   PLC/PLC Instance <-> EtherCAT Master BKCUCX/TcTerminals210_EK1100_1/TcTerminals210_1BK1250/A_0258(KM 2022, 16 Ch. Output (24V, 2.0 A))
//     PlcTask Outputs/GVL_iXlinker.EtherCAT_Master_BKCUCX.TcTerminals210_EK1100_1.TcTerminals210_1BK1250.A_0258_KM_2022_16_Ch_Output_24V_2_0_A.Channel_1.Output <-> Channel 1/Output
//     PlcTask Outputs/GVL_iXlinker.EtherCAT_Master_BKCUCX.TcTerminals210_EK1100_1.TcTerminals210_1BK1250.A_0258_KM_2022_16_Ch_Output_24V_2_0_A.Channel_2.Output <-> Channel 2/Output
//     PlcTask Outputs/GVL_iXlinker.EtherCAT_Master_BKCUCX.TcTerminals210_EK1100_1.TcTerminals210_1BK1250.A_0258_KM_2022_16_Ch_Output_24V_2_0_A.Channel_3.Output <-> Channel 3/Output
//     PlcTask Outputs/GVL_iXlinker.EtherCAT_Master_BKCUCX.TcTerminals210_EK1100_1.TcTerminals210_1BK1250.A_0258_KM_2022_16_Ch_Output_24V_2_0_A.Channel_4.Output <-> Channel 4/Output
//     PlcTask Outputs/GVL_iXlinker.EtherCAT_Master_BKCUCX.TcTerminals210_EK1100_1.TcTerminals210_1BK1250.A_0258_KM_2022_16_Ch_Output_24V_2_0_A.Channel_5.Output <-> Channel 5/Output
//     PlcTask Outputs/GVL_iXlinker.EtherCAT_Master_BKCUCX.TcTerminals210_EK1100_1.TcTerminals210_1BK1250.A_0258_KM_2022_16_Ch_Output_24V_2_0_A.Channel_6.Output <-> Channel 6/Output
//     PlcTask Outputs/GVL_iXlinker.EtherCAT_Master_BKCUCX.TcTerminals210_EK1100_1.TcTerminals210_1BK1250.A_0258_KM_2022_16_Ch_Output_24V_2_0_A.Channel_7.Output <-> Channel 7/Output
//     PlcTask Outputs/GVL_iXlinker.EtherCAT_Master_BKCUCX.TcTerminals210_EK1100_1.TcTerminals210_1BK1250.A_0258_KM_2022_16_Ch_Output_24V_2_0_A.Channel_8.Output <-> Channel 8/Output
//     PlcTask Outputs/GVL_iXlinker.EtherCAT_Master_BKCUCX.TcTerminals210_EK1100_1.TcTerminals210_1BK1250.A_0258_KM_2022_16_Ch_Output_24V_2_0_A.Channel_9.Output <-> Channel 9/Output
//     PlcTask Outputs/GVL_iXlinker.EtherCAT_Master_BKCUCX.TcTerminals210_EK1100_1.TcTerminals210_1BK1250.A_0258_KM_2022_16_Ch_Output_24V_2_0_A.Channel_10.Output <-> Channel 10/Output
//     PlcTask Outputs/GVL_iXlinker.EtherCAT_Master_BKCUCX.TcTerminals210_EK1100_1.TcTerminals210_1BK1250.A_0258_KM_2022_16_Ch_Output_24V_2_0_A.Channel_11.Output <-> Channel 11/Output
//     PlcTask Outputs/GVL_iXlinker.EtherCAT_Master_BKCUCX.TcTerminals210_EK1100_1.TcTerminals210_1BK1250.A_0258_KM_2022_16_Ch_Output_24V_2_0_A.Channel_12.Output <-> Channel 12/Output
//     PlcTask Outputs/GVL_iXlinker.EtherCAT_Master_BKCUCX.TcTerminals210_EK1100_1.TcTerminals210_1BK1250.A_0258_KM_2022_16_Ch_Output_24V_2_0_A.Channel_13.Output <-> Channel 13/Output
//     PlcTask Outputs/GVL_iXlinker.EtherCAT_Master_BKCUCX.TcTerminals210_EK1100_1.TcTerminals210_1BK1250.A_0258_KM_2022_16_Ch_Output_24V_2_0_A.Channel_14.Output <-> Channel 14/Output
//     PlcTask Outputs/GVL_iXlinker.EtherCAT_Master_BKCUCX.TcTerminals210_EK1100_1.TcTerminals210_1BK1250.A_0258_KM_2022_16_Ch_Output_24V_2_0_A.Channel_15.Output <-> Channel 15/Output
//     PlcTask Outputs/GVL_iXlinker.EtherCAT_Master_BKCUCX.TcTerminals210_EK1100_1.TcTerminals210_1BK1250.A_0258_KM_2022_16_Ch_Output_24V_2_0_A.Channel_16.Output <-> Channel 16/Output
//   PLC/PLC Instance <-> EtherCAT Master BKCUCX/TcTerminals210_EK1100_1/TcTerminals210_1BK1250/A_0259(KM 2042, 16 Ch. Output (24V, 0.5 A))
//     PlcTask Outputs/GVL_iXlinker.EtherCAT_Master_BKCUCX.TcTerminals210_EK1100_1.TcTerminals210_1BK1250.A_0259_KM_2042_16_Ch_Output_24V_0_5_A.Channel_1.Output <-> Channel 1/Output
//     PlcTask Outputs/GVL_iXlinker.EtherCAT_Master_BKCUCX.TcTerminals210_EK1100_1.TcTerminals210_1BK1250.A_0259_KM_2042_16_Ch_Output_24V_0_5_A.Channel_2.Output <-> Channel 2/Output
//     PlcTask Outputs/GVL_iXlinker.EtherCAT_Master_BKCUCX.TcTerminals210_EK1100_1.TcTerminals210_1BK1250.A_0259_KM_2042_16_Ch_Output_24V_0_5_A.Channel_3.Output <-> Channel 3/Output
//     PlcTask Outputs/GVL_iXlinker.EtherCAT_Master_BKCUCX.TcTerminals210_EK1100_1.TcTerminals210_1BK1250.A_0259_KM_2042_16_Ch_Output_24V_0_5_A.Channel_4.Output <-> Channel 4/Output
//     PlcTask Outputs/GVL_iXlinker.EtherCAT_Master_BKCUCX.TcTerminals210_EK1100_1.TcTerminals210_1BK1250.A_0259_KM_2042_16_Ch_Output_24V_0_5_A.Channel_5.Output <-> Channel 5/Output
//     PlcTask Outputs/GVL_iXlinker.EtherCAT_Master_BKCUCX.TcTerminals210_EK1100_1.TcTerminals210_1BK1250.A_0259_KM_2042_16_Ch_Output_24V_0_5_A.Channel_6.Output <-> Channel 6/Output
//     PlcTask Outputs/GVL_iXlinker.EtherCAT_Master_BKCUCX.TcTerminals210_EK1100_1.TcTerminals210_1BK1250.A_0259_KM_2042_16_Ch_Output_24V_0_5_A.Channel_7.Output <-> Channel 7/Output
//     PlcTask Outputs/GVL_iXlinker.EtherCAT_Master_BKCUCX.TcTerminals210_EK1100_1.TcTerminals210_1BK1250.A_0259_KM_2042_16_Ch_Output_24V_0_5_A.Channel_8.Output <-> Channel 8/Output
//     PlcTask Outputs/GVL_iXlinker.EtherCAT_Master_BKCUCX.TcTerminals210_EK1100_1.TcTerminals210_1BK1250.A_0259_KM_2042_16_Ch_Output_24V_0_5_A.Channel_9.Output <-> Channel 9/Output
//     PlcTask Outputs/GVL_iXlinker.EtherCAT_Master_BKCUCX.TcTerminals210_EK1100_1.TcTerminals210_1BK1250.A_0259_KM_2042_16_Ch_Output_24V_0_5_A.Channel_10.Output <-> Channel 10/Output
//     PlcTask Outputs/GVL_iXlinker.EtherCAT_Master_BKCUCX.TcTerminals210_EK1100_1.TcTerminals210_1BK1250.A_0259_KM_2042_16_Ch_Output_24V_0_5_A.Channel_11.Output <-> Channel 11/Output
//     PlcTask Outputs/GVL_iXlinker.EtherCAT_Master_BKCUCX.TcTerminals210_EK1100_1.TcTerminals210_1BK1250.A_0259_KM_2042_16_Ch_Output_24V_0_5_A.Channel_12.Output <-> Channel 12/Output
//     PlcTask Outputs/GVL_iXlinker.EtherCAT_Master_BKCUCX.TcTerminals210_EK1100_1.TcTerminals210_1BK1250.A_0259_KM_2042_16_Ch_Output_24V_0_5_A.Channel_13.Output <-> Channel 13/Output
//     PlcTask Outputs/GVL_iXlinker.EtherCAT_Master_BKCUCX.TcTerminals210_EK1100_1.TcTerminals210_1BK1250.A_0259_KM_2042_16_Ch_Output_24V_0_5_A.Channel_14.Output <-> Channel 14/Output
//     PlcTask Outputs/GVL_iXlinker.EtherCAT_Master_BKCUCX.TcTerminals210_EK1100_1.TcTerminals210_1BK1250.A_0259_KM_2042_16_Ch_Output_24V_0_5_A.Channel_15.Output <-> Channel 15/Output
//     PlcTask Outputs/GVL_iXlinker.EtherCAT_Master_BKCUCX.TcTerminals210_EK1100_1.TcTerminals210_1BK1250.A_0259_KM_2042_16_Ch_Output_24V_0_5_A.Channel_16.Output <-> Channel 16/Output
//   PLC/PLC Instance <-> EtherCAT Master BKCUCX/TcTerminals210_EK1100_1/TcTerminals210_1BK1250/A_0260(KM 2604, 4 Ch. Output Relay (230V AC/ 30V DC, 16A))
//     PlcTask Outputs/GVL_iXlinker.EtherCAT_Master_BKCUCX.TcTerminals210_EK1100_1.TcTerminals210_1BK1250.A_0260_KM_2604_4_Ch_Output_Relay_230V_AC_30V_DC_16A.Channel_1.Output <-> Channel 1/Output
//     PlcTask Outputs/GVL_iXlinker.EtherCAT_Master_BKCUCX.TcTerminals210_EK1100_1.TcTerminals210_1BK1250.A_0260_KM_2604_4_Ch_Output_Relay_230V_AC_30V_DC_16A.Channel_2.Output <-> Channel 2/Output
//     PlcTask Outputs/GVL_iXlinker.EtherCAT_Master_BKCUCX.TcTerminals210_EK1100_1.TcTerminals210_1BK1250.A_0260_KM_2604_4_Ch_Output_Relay_230V_AC_30V_DC_16A.Channel_3.Output <-> Channel 3/Output
//     PlcTask Outputs/GVL_iXlinker.EtherCAT_Master_BKCUCX.TcTerminals210_EK1100_1.TcTerminals210_1BK1250.A_0260_KM_2604_4_Ch_Output_Relay_230V_AC_30V_DC_16A.Channel_4.Output <-> Channel 4/Output
//   PLC/PLC Instance <-> EtherCAT Master BKCUCX/TcTerminals210_EK1100_1/TcTerminals210_1BK1250/A_0261(KM 2614, 4 Ch. Output Relay (230V AC/ 30V DC, 16A))
//     PlcTask Outputs/GVL_iXlinker.EtherCAT_Master_BKCUCX.TcTerminals210_EK1100_1.TcTerminals210_1BK1250.A_0261_KM_2614_4_Ch_Output_Relay_230V_AC_30V_DC_16A.Channel_1.Output <-> Channel 1/Output
//     PlcTask Outputs/GVL_iXlinker.EtherCAT_Master_BKCUCX.TcTerminals210_EK1100_1.TcTerminals210_1BK1250.A_0261_KM_2614_4_Ch_Output_Relay_230V_AC_30V_DC_16A.Channel_2.Output <-> Channel 2/Output
//     PlcTask Outputs/GVL_iXlinker.EtherCAT_Master_BKCUCX.TcTerminals210_EK1100_1.TcTerminals210_1BK1250.A_0261_KM_2614_4_Ch_Output_Relay_230V_AC_30V_DC_16A.Channel_3.Output <-> Channel 3/Output
//     PlcTask Outputs/GVL_iXlinker.EtherCAT_Master_BKCUCX.TcTerminals210_EK1100_1.TcTerminals210_1BK1250.A_0261_KM_2614_4_Ch_Output_Relay_230V_AC_30V_DC_16A.Channel_4.Output <-> Channel 4/Output
//   PLC/PLC Instance <-> EtherCAT Master BKCUCX/TcTerminals210_EK1100_1/TcTerminals210_1BK1250/A_0262(KM 2642, 2 Ch. Power Output Relay (230V AC/ 6A))
//     PlcTask Inputs/GVL_iXlinker.EtherCAT_Master_BKCUCX.TcTerminals210_EK1100_1.TcTerminals210_1BK1250.A_0262_KM_2642_2_Ch_Power_Output_Relay_230V_AC_6A.Channel_1.State_Relay <-> Channel 1/State Relay
//     PlcTask Inputs/GVL_iXlinker.EtherCAT_Master_BKCUCX.TcTerminals210_EK1100_1.TcTerminals210_1BK1250.A_0262_KM_2642_2_Ch_Power_Output_Relay_230V_AC_6A.Channel_2.State_Relay <-> Channel 2/State Relay
//     PlcTask Outputs/GVL_iXlinker.EtherCAT_Master_BKCUCX.TcTerminals210_EK1100_1.TcTerminals210_1BK1250.A_0262_KM_2642_2_Ch_Power_Output_Relay_230V_AC_6A.Channel_1.Output <-> Channel 1/Output
//     PlcTask Outputs/GVL_iXlinker.EtherCAT_Master_BKCUCX.TcTerminals210_EK1100_1.TcTerminals210_1BK1250.A_0262_KM_2642_2_Ch_Power_Output_Relay_230V_AC_6A.Channel_2.Output <-> Channel 2/Output
//   PLC/PLC Instance <-> EtherCAT Master BKCUCX/TcTerminals210_EK1100_1/TcTerminals210_1BK1250/A_0263(KM 2652, 2 Ch. Power Output Relay (230V AC/ 6A))
//     PlcTask Inputs/GVL_iXlinker.EtherCAT_Master_BKCUCX.TcTerminals210_EK1100_1.TcTerminals210_1BK1250.A_0263_KM_2652_2_Ch_Power_Output_Relay_230V_AC_6A.Channel_1.State_Auto <-> Channel 1/State Auto
//     PlcTask Inputs/GVL_iXlinker.EtherCAT_Master_BKCUCX.TcTerminals210_EK1100_1.TcTerminals210_1BK1250.A_0263_KM_2652_2_Ch_Power_Output_Relay_230V_AC_6A.Channel_2.State_Auto <-> Channel 2/State Auto
//     PlcTask Inputs/GVL_iXlinker.EtherCAT_Master_BKCUCX.TcTerminals210_EK1100_1.TcTerminals210_1BK1250.A_0263_KM_2652_2_Ch_Power_Output_Relay_230V_AC_6A.Channel_1.State_Relay <-> Channel 1/State Relay
//     PlcTask Inputs/GVL_iXlinker.EtherCAT_Master_BKCUCX.TcTerminals210_EK1100_1.TcTerminals210_1BK1250.A_0263_KM_2652_2_Ch_Power_Output_Relay_230V_AC_6A.Channel_2.State_Relay <-> Channel 2/State Relay
//     PlcTask Outputs/GVL_iXlinker.EtherCAT_Master_BKCUCX.TcTerminals210_EK1100_1.TcTerminals210_1BK1250.A_0263_KM_2652_2_Ch_Power_Output_Relay_230V_AC_6A.Channel_1.Output <-> Channel 1/Output
//     PlcTask Outputs/GVL_iXlinker.EtherCAT_Master_BKCUCX.TcTerminals210_EK1100_1.TcTerminals210_1BK1250.A_0263_KM_2652_2_Ch_Power_Output_Relay_230V_AC_6A.Channel_2.Output <-> Channel 2/Output
//   PLC/PLC Instance <-> EtherCAT Master BKCUCX/TcTerminals210_EK1100_1/TcTerminals210_1BK1250/A_0264(KM 2774-1001, 4 Ch. Blinds control, CM, Inputs (230V AC, 1A))
//     PlcTask Inputs/GVL_iXlinker.EtherCAT_Master_BKCUCX.TcTerminals210_EK1100_1.TcTerminals210_1BK1250.A_0264_KM_2774_1001_4_Ch_Blinds_control_CM_Inputs_230V_AC_1A.Channel_1.State <-> Channel 1/State
//     PlcTask Inputs/GVL_iXlinker.EtherCAT_Master_BKCUCX.TcTerminals210_EK1100_1.TcTerminals210_1BK1250.A_0264_KM_2774_1001_4_Ch_Blinds_control_CM_Inputs_230V_AC_1A.Channel_1.Data_In <-> Channel 1/Data In
//     PlcTask Outputs/GVL_iXlinker.EtherCAT_Master_BKCUCX.TcTerminals210_EK1100_1.TcTerminals210_1BK1250.A_0264_KM_2774_1001_4_Ch_Blinds_control_CM_Inputs_230V_AC_1A.Channel_1.Ctrl <-> Channel 1/Ctrl
//     PlcTask Outputs/GVL_iXlinker.EtherCAT_Master_BKCUCX.TcTerminals210_EK1100_1.TcTerminals210_1BK1250.A_0264_KM_2774_1001_4_Ch_Blinds_control_CM_Inputs_230V_AC_1A.Channel_1.Data_Out <-> Channel 1/Data Out
//   PLC/PLC Instance <-> EtherCAT Master BKCUCX/TcTerminals210_EK1100_1/TcTerminals210_1BK1250/A_0265(KM 2774, 4 Ch. Blinds control, CM, Inputs (230V AC, 1A))
